// TwinCAT 3 PLC project MagnetSystem_PI4
// ProgramVersion: 3.1.4023.0
// libraries:
//   CanItfHelper, * (Beckhoff Automation LLC)
//   Tc2_Math, * (Beckhoff Automation GmbH)
//   Tc2_Standard, * (Beckhoff Automation GmbH)
//   Tc2_System, * (Beckhoff Automation GmbH)
//   Tc2_TcpIp, * (Beckhoff Automation GmbH)
//   Tc2_Utilities, * (Beckhoff Automation GmbH)
//   Tc3_Module, * (Beckhoff Automation GmbH)
//   Tc3_EventLogger,3.1.30.0,Beckhoff Automation GmbH
// project tree:
//   DUTs/ E_Command.TcDUT, E_MagState.TcDUT (not stored), E_Status.TcDUT (not stored), ST_Alarm_Base.TcDUT, ST_canRxdata.TcDUT, ST_Coil_Base.TcDUT, ST_Coil_Ext_Analog1.TcDUT, ST_Control.TcDUT, ST_EngVal.TcDUT (not stored), ST_InstFeedback.TcDUT, ST_RecipeLocal.TcDUT, ST_Setpoints.TcDUT (not stored), ST_PermissivesToMainPLC.TcDUT, ST_Recipe.TcDUT (not stored), ST_SysParameters.TcDUT (not stored), ST_Trip_Base.TcDUT, ST_UC_Status.TcDUT (not stored), ST_UC_Status_Dummy.TcDUT (not stored), ST_UCDevices.TcDUT (not stored), ST_UC_Trip_Base.TcDUT (not stored)
//   GVLs/ Alarms_DB.TcGVL, Command.TcGVL, Devices.TcGVL (not stored), HMI_DB.TcGVL (not stored), Input.TcGVL (not stored), GVL.TcGVL (not stored), InstrumentReading.TcGVL (not stored), IO.TcGVL, MCP_IO.TcGVL (not stored), Output.TcGVL, Permissives_DB.TcGVL, Recipe.TcGVL, Setpoints.TcGVL (not stored), Trips_DB.TcGVL (not stored), Tx_Config.TcGVL
//   / PlcTask.TcTTO (not stored)
//   POUs/ ADC_10V.TcPOU (not stored), ADC_5V.TcPOU (not stored), Alias.TcPOU (not stored), AnalogConversion.TcPOU, CanInterface.TcPOU (not stored), CAN_comm.TcPOU (not stored), ChargeTimeCal.TcPOU, Delay2s.TcPOU (not stored), Graphs.TcPOU, Heartbeat.TcPOU, HMI.TcPOU, MAIN.TcPOU, MODE_SELECTION_1.TcPOU, Norm_x.TcPOU (not stored), Permissives.TcPOU, ChargeRlyClose_ChargerON_Seq.TcPOU (not stored), PWMO.TcPOU, Trips.TcPOU, Tx_MasterPLC.TcPOU (not stored), VoltageOutputCal.TcPOU
// real-time tasks:
//   TASK PlcTask: cycle T#10ms, priority 20, ADS port 350

// ---- DUTs/E_Command.TcDUT
{attribute 'qualified_only'}
{attribute 'strict'}
{attribute 'to_string'}
//Command from Master PLC
TYPE E_Command :
(
	//Requested Magnetic State
	FULL_SHUTDOWN 	:= 0, 
	IDLE			:= 1, 
	CHARGE			:= 3, 
	//PAUSE_CHARGE	:= 4, //no need to use pause charge
	SHOOT			:= 6, 
	//SHUTDOWN		:= 8, //remove
	DUMP			:= 9
);
END_TYPE

// ---- DUTs/ST_Alarm_Base.TcDUT
TYPE ST_Alarm_Base :
STRUCT
(*
	AI_CH1_UnderVoltage		: BOOL;
	AI_CH1_OverVoltage		: BOOL;
	AI_CH1_belowLIM1		: BOOL;
	AI_CH1_aboveLIM1		: BOOL;
	
	AI_CH2_UnderVoltage		: BOOL;
	AI_CH2_OverVoltage		: BOOL;
	AI_CH2_belowLIM1		: BOOL;
	AI_CH2_aboveLIM1		: BOOL;
	
	AI_CH3_UnderVoltage		: BOOL;
	AI_CH3_OverVoltage		: BOOL;
	AI_CH3_belowLIM1		: BOOL;
	AI_CH3_aboveLIM1		: BOOL;
	
	ChargerVoltageReading_Faulted	: BOOL;
	CurrentReading_Faulted		 	: BOOL;
	BfieldReading_Faulted			: BOOL;
*)
	AlarmWord : WORD;
END_STRUCT
END_TYPE

// ---- DUTs/ST_canRxdata.TcDUT
TYPE ST_canRxdata :
STRUCT
	cobID			: STRING;
	deviceID		: ARRAY [1..10] OF STRING; // will make it 1..10 later
	byteData		: ARRAY [0..7] OF USINT;
	byteData_hexstr	: ARRAY [0..7] OF STRING;
END_STRUCT
END_TYPE

// ---- DUTs/ST_Coil_Base.TcDUT
//Base coil type with all the Common functionality
TYPE ST_Coil_Base :
STRUCT
	afterShot_actualCoilCurrent_WaveForm	: WORD;
	requiredTimeToCharge					: TIME;
	measuredMagneticField					: DINT;
		
	ChargeVoltageFeedback					: REAL;
	ChargeVoltageFeedback_raw				: INT;
	ChargerVoltageFeedback_norm				: REAL;
	TotalVoltage							: REAL;
	
	CurrentFeedback							: REAL;
	CurrentFeedback_raw						: INT;
	CurrentFeedback_norm					: REAL;

	Measured_Bfield							: REAL;
	Measured_Bfield_raw						: INT;
	B_fieldFeedback_norm					: REAL;
	
	chargerSetpoint							: INT;  //0-100% analog PWM 24V output -> (0 - 10V)
	chargerSetpoint_norm					: REAL;
	chargerSetpoint_raw						: REAL;
	currentSetpoint							: INT;  //0-100% analog PWM 24V output -> (0.5 - 4.5V)
	currentSetpoint_norm					: REAL;
	currentSetpoint_raw						: REAL;
	//currentSetpointFromMaster: REAL;

	PSU0_active								: BOOL := FALSE;
	PSU1_DCOK								: BOOL;
	Local_StopPB_Pressed					: BOOL;  //NC
	DumpRelay1_closed						: BOOL;
	DumpRelay2_closed						: BOOL;
	ChargeRelay_closed						: BOOL := FALSE;
	ChargerIsEnabled						: BOOL := FALSE; //feedback from charger
	FlybackD1_Alive							: BOOL := FALSE;
	FlybackD2_Alive							: BOOL := FALSE;
	
	DumpResistorTemperatureHigh				: BOOL; 
	GroundLoopCurrentDetected				: BOOL;
	CoilTemperatureHigh						: BOOL := FALSE;
	AC_Interlock_RlyClose					: BOOL;
	LossPneumaticPressure					: BOOL;
	
	OpenDumpRelays							: BOOL := FALSE;
	closeChargeRelay						: BOOL := FALSE;
	enableOutputToCharger					: BOOL := FALSE;  //output going to charger
	CloseACInterlockRly						: BOOL := FALSE;
	SystemFaulted							: BOOL := FALSE;
	SystemCharging							: BOOL := FALSE;
	SystemReady								: BOOL := FALSE;
	CloseHVisolationRelay					: BOOL; //relay 6 (24vdc) to control relay 7 & 8 (two 120vac ross relays)
	HVisolationRelayClosed					: BOOL;
	OutputRelayOpen							: BOOL;
	
	CoilEnabled								: BOOL := TRUE;
	AllCapsCharged							: BOOL;
	NumOfCap								: INT := 4;
	
	//CoilSafetyOK							: BOOL;
	CapWarning								: BOOL;  //comes from UltraCaps CANBUS message
	CapAlarm								: BOOL;
	CapVoltage								: ARRAY[1..15] OF INT;   //Comes from UlgraCaps CANBUS message
	CapCellTemp								: ARRAY[1..15] OF INT;
	
	ChargerVoltageFault_TON : TON;
	ChargerVoltageFault_ET : TIME;
	CurrentSensorFault_TON : TON;
	CurrentSensorFault_ET : TIME;
	BfieldSensorFault_TON : TON;
	BfieldSensorFault_ET : TIME;
	
	//CAN_id: INT;
	//CAN_AdsAddr: AMSADDR;
	//CAN_netID: AMSNETID;
	//CAN_port: WORD;
	//CAN_error: USINT;
	//CAN_State: UINT;
	//CAN_RxErrorCounter: USINT;	
	//CAN_TxErrorCounter: USINT;	
	//CAN_DiagFlag: BOOL;
	
	//UltraCap_CAN_ID : STRING;
	UltraCap			: ARRAY[1..10] OF  ST_UC_Status;  //assuming 10 uc in one coil
	UltraCap_Dummy		: ST_UC_Status_Dummy; //buffer temp for uc 7f
	UC_Dummy_ID_hexstr	: STRING;
	
	CanTx_config_ID 	: UDINT;
	CanTx_config_length : UINT;
	CanTx_config_request: ARRAY[0..7] OF BYTE;
		
END_STRUCT
END_TYPE

// ---- DUTs/ST_Coil_Ext_Analog1.TcDUT
TYPE ST_Coil_Ext_Analog1 EXTENDS ST_Coil_Base :
STRUCT
	iAnalogOfWinning : INT;
END_STRUCT
END_TYPE

// ---- DUTs/ST_Control.TcDUT
TYPE ST_Control :
STRUCT
	ClearAllFault : BOOL;
	Abort		  : BOOL;
END_STRUCT
END_TYPE

// ---- DUTs/ST_InstFeedback.TcDUT
TYPE ST_InstFeedback :
STRUCT
	ChargerVolt : REAL;
	CapVolt		: ARRAY [1..15] OF REAL;
	Cur  		: REAL;
	TotalVoltage: REAL;
END_STRUCT
END_TYPE

// ---- DUTs/ST_RecipeLocal.TcDUT
TYPE ST_RecipeLocal :
STRUCT
	chargerSetpoint 	: INT;  
	currentSetpoint 	: INT;   
	CurrentDuration		: TIME;   
END_STRUCT
END_TYPE

// ---- DUTs/ST_PermissivesToMainPLC.TcDUT
TYPE ST_PermissivesToMainPLC :
STRUCT
	ChargePermOK			: BOOL;
	ShootPermOK				: BOOL;
	
	AlldcPSUok				: BOOL;
	AllacInterlock_Closed	: BOOL;
	All_Coil_TemperatureOK	: BOOL;
	AllDumpResistorTempOK	: BOOL;
	NoGroundLoopCurrentDetected: BOOL;
	//AllFlybackDiodes_Alive	: BOOL;
	AllChargerEnabled		: BOOL;
	AnyCoilDisabled 		: BOOL;		
	SafetyOK				: BOOL;
	AllDumpRelayOpen		: BOOL;
	AllChargerRelay_Closed	: BOOL;
	AdminFaultBypassOn		: BOOL;
	// voltage feedback from CANbus to main plc
	
END_STRUCT
END_TYPE

// ---- DUTs/ST_Trip_Base.TcDUT
TYPE ST_Trip_Base :
STRUCT
	ChargerVoltageReadingFaulted 		: BOOL;
	CurrentReadingFaulted 		 		: BOOL;
	BfieldReadingFaulted 		 		: BOOL;
	
	ACInterlockRelayFailedtoClose		: BOOL;
	ACInterlockRelayFailedtoOpen 		: BOOL;
	ACintLockRlyCloseFaultDelay_TON		: TON;
	ACintLockRlyOpenFaultDelay_TON		: TON;
	
	DumpRelay1_FailtoClose		 		: BOOL;
	DumpRelay1_FailtoOpen		 		: BOOL;
	DumpRlyCloseFaultDelay_TON 		 	: TON;
	DumpRlyOpenFaultDelay_TON 		 	: TON;
	
	DumpRelay2_FailtoClose		 : BOOL;
	DumpRelay2_FailtoOpen		 : BOOL;
	
	ChargeRelay_FailtoClose		 : BOOL;
	ChargeRelay_FailtoOpen		 : BOOL;
	ChrgRlyCloseFaultDelay_TON	 : TON;
	ChrgRlyOpenFaultDelay_TON	 : TON;
	
	
	HVisoRelayFailedToOpen		: BOOL;
	HVRelayOpenFaultDelay_TON	: TON;
	HVisoRelayFailedToClose		: BOOL;
	HVRelayCloseFaultDelay_TON	: TON;
	
	UltraCap					: ARRAY[1..10] OF ST_UC_Trip_Base;
	AnyCapOverV_warning			: BOOL;  //cell voltage > 2.85V - warning, > 2.9V - alarm
	AnyCapOverV_alarm			: BOOL;  //cell voltage > 2.85V - warning, > 2.9V - alarm
	AnyCapOverTemp_warning		: BOOL; //cell >50C - warning, >60C - alarm
	AnyCapOverTemp_alarm		: BOOL; //cell >50C - warning, >60C - alarm
END_STRUCT
END_TYPE

// ---- GVLs/Alarms_DB.TcGVL
{attribute 'qualified_only'}
VAR_GLOBAL
	Coil1 : ST_Alarm_Base;
	Coil2 : ST_Alarm_Base;
	Coil3 : ST_Alarm_Base;
	Coil4 : ST_Alarm_Base;
	Coil5 : ST_Alarm_Base;
	Coil6 : ST_Alarm_Base;
	Coil7 : ST_Alarm_Base;
	Coil8 : ST_Alarm_Base;
	Coil9 : ST_Alarm_Base;
	Coil10 : ST_Alarm_Base;
	
	AlarmWord_11 : ST_Alarm_Base;
	AlarmWord_22 : ST_Alarm_Base;
	AlarmWord_23 : ST_Alarm_Base;
	AlarmWord_24 : ST_Alarm_Base;
	AlarmWord_25 : ST_Alarm_Base;
	AlarmWord_26 : ST_Alarm_Base;
	AlarmWord_27 : ST_Alarm_Base;
	AlarmWord_88 : ST_Alarm_Base;
END_VAR

// ---- GVLs/Command.TcGVL
{attribute 'qualified_only'}
VAR_GLOBAL

	eCommand : E_Command;
END_VAR

// ---- GVLs/IO.TcGVL
{attribute 'qualified_only'}
VAR_GLOBAL
	//PB01_Rx AT%I* : ARRAY [0..145] OF BYTE;
	//PB01_Tx AT%Q* : ARRAY [0..145] OF BYTE;
END_VAR

// ---- GVLs/Output.TcGVL
{attribute 'qualified_only'}
VAR_GLOBAL
//LCP 1	
	//EL2502 - PWM Output
	R2_02_00 AT %Q*: INT;
	R2_02_01 AT %Q*: INT;
	
	// EL 2008 - DQ
	R2_05_00 AT %Q*: BOOL;
	R2_05_01 AT %Q*: BOOL;
	R2_05_02 AT %Q*: BOOL;
	R2_05_03 AT %Q*: BOOL;
	R2_05_04 AT %Q*: BOOL;
	R2_05_05 AT %Q*: BOOL;
	R2_05_06 AT %Q*: BOOL;
	R2_05_07 AT %Q*: BOOL; //spare
	
	R2_06_CANrequest AT %Q*: EXTCANQUEUE;
//LCP 2	***********************************************
	//EL2502 - PWM Output
	R3_02_00 AT %Q*: INT;
	R3_02_01 AT %Q*: INT;
	
	// EL 2008 - DQ
	R3_05_00 AT %Q*: BOOL;
	R3_05_01 AT %Q*: BOOL;
	R3_05_02 AT %Q*: BOOL;
	R3_05_03 AT %Q*: BOOL;
	R3_05_04 AT %Q*: BOOL;
	R3_05_05 AT %Q*: BOOL;
	R3_05_06 AT %Q*: BOOL;
	R3_05_07 AT %Q*: BOOL; //spare
	
	R3_06_CANrequest AT %Q*: EXTCANQUEUE;	
END_VAR

// ---- GVLs/Permissives_DB.TcGVL
{attribute 'qualified_only'}
VAR_GLOBAL
	ChargePermOK			: BOOL;
	ShootPermOK				: BOOL;
	//AllChargers_Active		: BOOL;
	AlldcPSUok				: BOOL;
	AllacInterlock_Closed	: BOOL;
	All_Coil_TemperatureOK	: BOOL;
	AllDumpResistorTempOK	: BOOL;
	NoGroundLoopCurrentDetected: BOOL;
	//AllFlybackDiodes_Alive	: BOOL;
	AllChargerEnabled		: BOOL;
	AnyCoilDisabled 		: BOOL;		
	SafetyOK				: BOOL;
	AllDumpRelayOpen		: BOOL;
	//AllDumpRelayClose		: BOOL;
	AllChargerRelay_Closed	: BOOL;
	AllCoilCapsCharged		: BOOL;
	NoPneumaticPressureLoss : BOOL;
END_VAR

// ---- GVLs/Recipe.TcGVL
{attribute 'qualified_only'}
VAR_GLOBAL
	Coil : ARRAY[1..10] OF ST_Recipe;
	General : ST_Recipe;
END_VAR

// ---- GVLs/Tx_Config.TcGVL
{attribute 'qualified_only'}
VAR_GLOBAL
	CoilSP : ARRAY[1..10] OF ST_Setpoints;
	
	ReadyToChargeRunOutTime	: REAL;
	ChargingRunOutTime		: REAL;
	ChargePausedRunOutTime	: REAL;
	ReadyToShootRunOutTime	: REAL;				
	ShootingRunOutTime		: REAL;
	PostShotRunOutTime		: REAL;
	DumpingRunOutTime		: REAL;
	CoilInst				: ARRAY[1..10] OF ST_InstFeedback;
	
END_VAR

// ---- POUs/AnalogConversion.TcPOU
PROGRAM AnalogConversion
VAR	
	i : INT  := 1;
	
END_VAR

//*******************Output Sepoints come from the Screen room recipe, the sysparameters would need to mapped here******//
//ie Setpoints.coil[1].engval.max_chargervoltage := Recipe.
Devices.Coil[1].NumOfCap := Setpoints.Coil[1].SysParameters.NumOfCaps;


//Converting raw data into Voltage Reading (0-10V), (0.5-4.5V)

//LCP1
// Voltage feedback - 10V = Max voltage (102V)
Devices.Coil[1].ChargerVoltageFeedback_norm := Norm_x (raw_input := INT_TO_REAL(Devices.Coil[1].ChargeVoltageFeedback_raw),
										x_max := 32767,
										x_min := 0);
										
InstrumentReading.R2_01_CH00 := Devices.Coil[1].ChargerVoltageFeedback_norm * 10;

//Charger Voltage = (max voltage - min voltage) * measured_voltage / range(voltage)
Devices.Coil[1].ChargeVoltageFeedback := (Setpoints.Coil[1].EngVal.Max_chargerVoltage - Setpoints.Coil[1].EngVal.Min_chargerVoltage) * ADC_10V (normal_input := Devices.Coil[1].ChargerVoltageFeedback_norm,
																					x_max := 10,
																					x_min := 0);

//Current feedback - 4.5V = 600Amp????
Devices.Coil[1].CurrentFeedback_norm := Norm_x (raw_input := INT_TO_REAL(Devices.Coil[1].CurrentFeedback_raw),
								x_max := 32767*4.5/10,
								x_min := 32767*0.5/10);
						
InstrumentReading.R2_01_CH01 := Devices.Coil[1].CurrentFeedback_norm * (4.5-0.5);

//Current feedback for each ultracap
Devices.Coil[1].CurrentFeedback := (Setpoints.Coil[1].EngVal.Max_current_perCap - Setpoints.Coil[1].EngVal.Min_current_perCap) * ADC_5V (normal_input := Devices.Coil[1].CurrentFeedback_norm,
																								x_max := 4.5,
																								x_min := 0.5);

//CurrentFeedback_norm := Norm_x (raw_input := INT_TO_REAL(Input.R2_01_01), x_max := 32767*4.5/10, x_min := 32767*0.5/10);
//coil1.CurrentFeedback := CurrentFeedback_norm * 4;

//B-field - (0-10V) 10V = ?? Tesla
Devices.Coil[1].B_fieldfeedback_norm := Norm_x (raw_input := INT_TO_REAL(Devices.Coil[1].Measured_Bfield_raw),
								x_max := 32767,
								x_min := 0);
								
InstrumentReading.R2_01_CH02 := Devices.Coil[1].B_fieldfeedback_norm * 10;

//Charger Voltage = (max voltage - min voltage) * measured_voltage / range(voltage)
Devices.Coil[1].Measured_Bfield := (Setpoints.Coil[1].EngVal.Max_Tesla - Setpoints.Coil[1].EngVal.Min_Tesla) * ADC_10V(normal_input := Devices.Coil[1].B_fieldfeedback_norm,
																x_max := 10,
																x_min := 0);

																
//PWM Output

//set limits of charger voltage input 
FOR i := 1 TO 10 BY 1 DO
	IF Devices.Coil[i].chargerSetpoint >= REAL_TO_INT (Setpoints.Coil[1].EngVal.Max_chargerVoltage) THEN
		Devices.Coil[i].chargerSetpoint := REAL_TO_INT (Setpoints.Coil[1].EngVal.Max_chargerVoltage);
	END_IF;
	//This should never happend
	IF Devices.Coil[i].chargerSetpoint_raw >= (10/24 * 32767) THEN
		Devices.Coil[i].chargerSetpoint_raw := (10/24 * 32767);
	END_IF;
END_FOR;

Devices.Coil[1].chargerSetpoint_norm := Norm_x (raw_input := INT_TO_REAL (Devices.Coil[1].chargerSetpoint), 
												x_max := Setpoints.Coil[1].EngVal.Max_chargerVoltage,
												x_min := Setpoints.Coil[1].EngVal.Min_chargerVoltage);

Devices.Coil[1].chargerSetpoint_raw := PWMO (norm_input := Devices.Coil[1].chargerSetpoint_norm, 
												x_max := 24,
												x_min := 0); 	


//Current set point output
//set limits of charger voltage input 
FOR i := 1 TO 10 BY 1 DO
	IF Devices.Coil[i].currentSetpoint >= REAL_TO_INT (Setpoints.Coil[1].EngVal.Max_current_perCap) THEN
		Devices.Coil[i].currentSetpoint := REAL_TO_INT (Setpoints.Coil[1].EngVal.Max_current_perCap);
	END_IF;
	//This should never happend - Current setpoint board takes 0.5V - 4.5V
	IF Devices.Coil[i].currentSetpoint_raw >= (4.5/24 * 32767) THEN
		Devices.Coil[i].currentSetpoint_raw := (4.5/24 * 32767);
	END_IF;
END_FOR;

Devices.Coil[1].currentSetpoint_norm := Norm_x (raw_input := INT_TO_REAL (Devices.Coil[1].currentSetpoint), 
												x_max := Setpoints.Coil[1].EngVal.Max_current_perCap,
												x_min := Setpoints.Coil[1].EngVal.Min_current_perCap);
//current output for each cap
Devices.Coil[1].currentSetpoint_raw := PWMO (norm_input := Devices.Coil[1].currentSetpoint_norm, 
												x_max := 24,
												x_min := 0); 	


//uncomment this when PWM output module is ready.											
(*
//LCP1
Output.R2_02_00 := Devices.Coil[1].chargerSetpoint_raw; 
Output.R2_02_01 := Devices.Coil[1].currentSetpoint_raw;

//LCP2
Output.R3_02_00 := Devices.Coil[2].chargerSetpoint_raw; 
Output.R3_02_01 := Devices.Coil[2].currentSetpoint_raw;
*)

//reset counter
IF i > 10 THEN
	i:=1;
END_IF;

END_PROGRAM

// ---- POUs/PWMO.TcPOU
FUNCTION PWMO : INT
VAR_INPUT
	Norm_input : REAL;
	x_max : REAL := 24;
	x_min : REAL := 0;
END_VAR
VAR
	voltage_reading : REAL;
END_VAR

voltage_reading := 10 * Norm_input;
PWMO := REAL_TO_INT (32767 * (voltage_reading - x_min) / (x_max - x_min));

END_FUNCTION

// ---- POUs/ChargeTimeCal.TcPOU
FUNCTION_BLOCK ChargeTimeCal
VAR_INPUT
	I_setpoint 	: REAL := 400;
	t_duration	: REAL := 4;
	NumOfCaps	: REAL := 15;
	C_percap	: REAL := 88;
	VMAXperCap	: REAL := 100;
	R_coil		: REAL := 1.1;
	L_coil		: REAL := 0.5;
	VMAXcharger	: REAL := 1500;
	Pcharger	: REAL := 15000;
	NumOfCharger: REAL := 4;
END_VAR
VAR_OUTPUT
	Tuntilfullcharge	: REAL;
END_VAR
VAR
	V_chargerCC2CP : REAL;
	C_total		   : REAL;
	V_capsmax	   : REAL;
	E_resistivepulse : REAL;
	E_inductivepulse : REAL;
	E_pulse			 : REAL;
	VchrSPrequested  : REAL;
	VchrSPactual     : REAL;
	I_peakchargecurrent : REAL;
	Icc					: REAL;
	Icp					: REAL;
	Vpresent			: REAL;
	Vfinal				: REAL;
	VpresentCC			: REAL;
	VfinalCC			: REAL;
	Tcc					: REAL;
	VpresentCP			: REAL;
	Tcp					: REAL;
END_VAR

V_chargerCC2CP := VMAXcharger / 2;

C_total := C_percap/NumOfCaps;
V_capsmax := VMAXpercap * NumOfCaps;
E_resistivepulse := LREAL_TO_REAL(EXPT(I_setpoint, 2))*R_coil*t_duration;
E_inductivepulse := L_coil * LREAL_TO_REAL(EXPT(I_setpoint, 2))/2;
E_pulse := E_resistivepulse + E_inductivepulse;
VchrSPrequested := SQRT(2*E_pulse/C_total);

IF VchrSPrequested > V_capsmax THEN
	VchrSPactual := V_capsmax;
	ELSE
		VchrSPactual := VchrSPrequested;	
END_IF

//I_peakchargecurrent := Pcharger * NumOfCharger / (2*VMAXcharger);
I_peakchargecurrent := Pcharger * NumOfCharger * 2 / VMAXcharger;
Icc := I_peakchargecurrent;
Icp := I_peakchargecurrent * (0.5 + ((VMAXcharger - Vpresent)/VMAXcharger));
Vfinal := 1400; //hard coded???
VpresentCC := 200; // hard coded???

IF Vfinal > V_chargerCC2CP THEN
	VfinalCC := V_chargerCC2CP;
	ELSIF Vfinal < V_chargerCC2CP THEN
		VfinalCC := Vfinal;
END_IF

Tcc := (V_chargerCC2CP - VpresentCC)*C_total/I_peakchargecurrent;

VpresentCP := V_chargerCC2CP;
Tcp := -((VMAXcharger*C_total)/I_peakchargecurrent)*LN((1.5*VMAXcharger-Vfinal)/(1.5*VMAXcharger-VpresentCP));

Tuntilfullcharge := Tcc + Tcp;

END_FUNCTION_BLOCK

// ---- POUs/Graphs.TcPOU
PROGRAM Graphs
VAR
	i : INT :=0;
	coil1_current: ARRAY[1..1, 1..100] OF REAL;
	//coil1_current : ARRAY	

END_VAR

// still need more work

FOR i := 1 TO 100 DO 
	coil1_current[1, i] := Devices.coil1.CurrentFeedback;
	
END_FOR

FOR i := 100 TO 2 BY -1 DO
	coil1_current[1, i-1] := Devices.coil1.CurrentFeedback;
END_FOR

IF coil1_current[1, 1] = 100 THEN
	i := -1;
ELSIF coil1_current[1, 1] = 1 THEN
	i := 1;
END_IF

END_PROGRAM

// ---- POUs/Heartbeat.TcPOU
PROGRAM Heartbeat
VAR
	start_TON				: TON;
	start_TON_et 			: TIME;
	reset_TON 				: TON;
	reset_TON_et 			: TIME;
	screen_refresh_pulse 	: BOOL;
	
	pulse_1Hz_Start_TON		: TON;
	pulse_1Hz_Start_PT		: TIME := T#4MS;
	pulse_1Hz_Reset_TON		: TON;
	pulse_1Hz_Reset_PT		: TIME := T#6MS;
	pulse_1Hz				: BOOL;
END_VAR

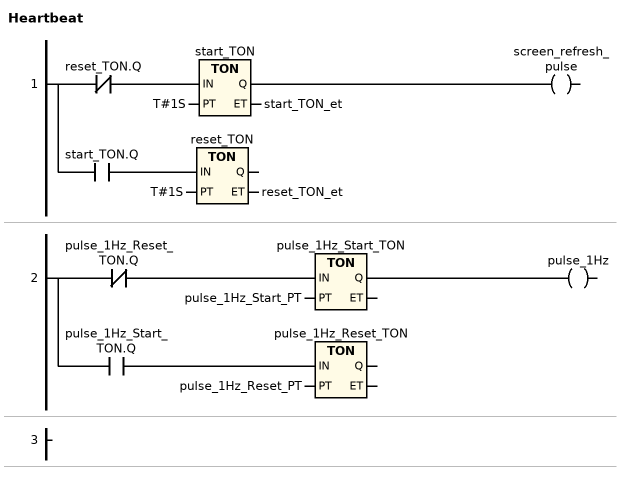
// NETWORK 1
start_TON(IN := NOT reset_TON.Q, PT := T#1S, ET => start_TON_et); // TON
screen_refresh_pulse := start_TON.Q;
reset_TON(IN := start_TON.Q, PT := T#1S, ET => reset_TON_et); // TON

// NETWORK 2
pulse_1Hz_Start_TON(IN := NOT pulse_1Hz_Reset_TON.Q, PT := pulse_1Hz_Start_PT); // TON
pulse_1Hz := pulse_1Hz_Start_TON.Q;
pulse_1Hz_Reset_TON(IN := pulse_1Hz_Start_TON.Q, PT := pulse_1Hz_Reset_PT); // TON

// NETWORK 3

END_PROGRAM

// ---- POUs/HMI.TcPOU
PROGRAM HMI
VAR
END_VAR



HMI_DB.ReadyToChargeRunOutTime	:= TIME_TO_DINT (MODE_SELECTION_1.ReadyToChargeRunOutTMR_PT - MODE_SELECTION_1.ReadyToChargeRunOutTMR_TON.ET)/1000;
HMI_DB.ChargingRunOutTime		:= TIME_TO_DINT (MODE_SELECTION_1.ChargingRunOutTMR_PT - MODE_SELECTION_1.ChargingRunOutTMR_TON.ET)/1000;	
HMI_DB.ChargePausedRunOutTime	:= TIME_TO_DINT (MODE_SELECTION_1.ChargePausedRunOutTMR_PT - MODE_SELECTION_1.ChargePausedRunOutTMR_ET)/1000;	
HMI_DB.ReadyToShootRunOutTime	:= TIME_TO_DINT (MODE_SELECTION_1.ReadyToShootRunOutTMR_PT - MODE_SELECTION_1.ReadyToShootRunOutTMR_ET)/1000;					
HMI_DB.ShootingRunOutTime		:= TIME_TO_DINT (MODE_SELECTION_1.ShootingRunOutTMR_PT - MODE_SELECTION_1.ShootingRunOutTMR_ET)/1000;			
HMI_DB.PostShotRunOutTime		:= TIME_TO_DINT (MODE_SELECTION_1.PostShotRunOutTMR_PT - MODE_SELECTION_1.PostShotRunOutTMR_ET)/1000;			
HMI_DB.DumpingRunOutTime		:= TIME_TO_DINT (MODE_SELECTION_1.DumpingRunOutTMR_PT - MODE_SELECTION_1.DumpingRunOutTMR_ET)/1000;

END_PROGRAM

// ---- POUs/MODE_SELECTION_1.TcPOU
PROGRAM MODE_SELECTION_1
VAR
	//MagnetState : (FULL_SHUTDOWN, IDLE, READY_TO_CHARGE, CHARGING, CHARGING_PAUSED, READY_TO_SHOOT, SHOOTING, POST_SHOT, SHUTDOWN, DUMPING); 
	eMagState : E_MagState := 0;
	//bChargingDone: BOOL;
	eCommand : E_Command; // Requested State (FULL_SHUT_DOWN = 0, IDLE = 1, CHARGE = 2, CHARGE_PAUSED, SHOOT = 3, POST_SHOT = 4, SHUTDOWN = 5, DUMPING = 6)
	eStatus : E_Status; // Actual Status (FULL_SHUTDOWN = 0, IDLE = 1, READY_TO_CHARGE = 2, CHARGE = 3, CHARGE_PAUSED = 4, READY_TO_SHOOT = 5, SHOOTING = 6, POST_SHOT = 7, SHUTDOWN = 8, DUMPING = 9, TRIPPED = 10, MANUAL_MODE = 11)
	i: INT;
	
	ChargerOFF_ChrgRlyOPEN_Delay_FShutDown_TON	: TON;
	timerBTW_ChrgRly_ChrgEnable_ChrgPause_TON	: TON;
	timerBTW_ChrgRly_ChrgEnable_ReadyToShoot_TON: TON;
	
	timerBTW_ChrgRly_ChrgEnable_Chrging_TON		: TON;
	timerBTW_ChrgRly_ChrgEnable_PT 	: TIME := T#500MS;
	timerBTW_ChrgRly_ChrgEnable_ET  : TIME;
	
	timerBTW_DUMP_IDLE 				: TON;
	timerBTW_DUMP_IDLE_PT 			: TIME := T#15S;
	timerBTW_DUMP_IDLE_ET 			: TIME;
	
	timerForChargertoTurnOn_TON		: TON;
	timerForChargertoTurnOn_PT		: TIME := T#10S;
	timerForChargertoTurnOn_ET		: TIME;
	ChargersReady					: BOOL;
	
	timerBTW_Shoot_PostShot_TON		: TON;
	timerBTW_Shoot_PostShot_PT      : TIME := T#2S;
	timerBTW_Shoot_PostShot_ET		: TIME;
	
	timerBTW_ChrgEnable_ChrgRly_ShutDown_TON	: TON;
	timerBTW_ChrgEnable_ChrgRly_PT				: TIME := T#1S;
	timerBTW_ChrgEnable_ChrgRly_ET				: TIME;
	
	timerBTW_ChrgEnable_ChrgRly_Dumping_TON		: TON;
	timerBTW_ChrgEnable_ChrgRly_Dumping_ET		: TIME;
	
	timerBTW_ChrgEnable_ChrgRly_Tripped_TON		: TON;
	timerBTW_ChrgEnable_ChrgRly_Tripped_ET		: TIME;
	
	ReadyToChargeRunOutTMR_TON					: TON;
	ReadyToChargeRunOutTMR_PT					: TIME := T#1200S;
	ReadyToChargeRunOutTMR_ET					: TIME;
	
	ChargePausedRunOutTMR_TON					: TON;
	ChargePausedRunOutTMR_PT					: TIME := T#30S;
	ChargePausedRunOutTMR_ET					: TIME;
	
	ReadyToShootRunOutTMR_TON					: TON;
	ReadyToShootRunOutTMR_PT					: TIME := T#60S;
	ReadyToShootRunOutTMR_ET					: TIME;
	
	ShootingRunOutTMR_TON						: TON;
	ShootingRunOutTMR_PT						: TIME := T#3S;
	ShootingRunOutTMR_ET						: TIME;
	
	PostShotRunOutTMR_TON						: TON;
	PostShotRunOutTMR_PT						: TIME := T#2S;
	PostShotRunOutTMR_ET						: TIME;
	
	DumpingRunOutTMR_TON						: TON;
	DumpingRunOutTMR_PT							: TIME := T#300S;
	DumpingRunOutTMR_ET							: TIME;
	
	ChargingRunOutTMR_TON						: TON;
	ChargingRunOutTMR_PT						: TIME := T#600S;
	ChargingRunOutTMR_ET						: TIME;
	
	stControl									: ST_Control;
END_VAR


//LCP Indicator for charged/charging
FOR i := 1 TO 10 BY 1 DO
	IF ( Devices.Coil[i].ChargeRelay_closed = TRUE AND 
		Devices.Coil[i].CoilEnabled = TRUE AND 
		Devices.Coil[i].enableOutputToCharger = TRUE ) OR Devices.Coil[i].ChargeVoltageFeedback >= 10
	THEN
		Devices.Coil[i].SystemCharging := TRUE;
		ELSE
			Devices.Coil[i].SystemCharging := FALSE;
	END_IF;
END_FOR;

//IF any one of the systems is charging or charge, then all system discharge is false, otherwise true
IF Devices.Coil[i].SystemCharging = TRUE THEN
	GVL.AllSystemsDischarged := FALSE;
ELSE
	GVL.AllSystemsDischarged := TRUE;
END_IF;

// IF system is tripped at anytime, it goes to tripped state
IF Trips_DB.SystemTripped = TRUE OR Permissives_DB.SafetyOK = FALSE THEN
	eMagState := E_MagState.TRIPPED;
END_IF;

IF MCP_IO.RemoteModeSelected = FALSE OR HMI_DB.RemoteModeSelected = FALSE THEN  //change auto to remote / manu to local
	eStatus := E_Status.MANUAL_MODE;
END_IF

//At any point, if screen room ask to dump, it goes to dump state
IF (MCP_IO.RemoteModeSelected = TRUE AND eCommand = E_Command.DUMP) OR stControl.Abort = TRUE THEN
	eMagState := E_Magstate.DUMPING;
END_IF;

FOR i := 1 TO 10 BY 1 DO
	Devices.Coil[i].NumOfCap := Tx_Config.CoilSP[i].SysParameters.NumOfCaps;
END_FOR


//Process Starts
CASE eMagState OF 
	//Full Shutdown
	E_MagState.FULL_SHUTDOWN:
						//Disable all Chargers
						FOR i := 1 TO 10 BY 1 DO
							
							//open (de-energize) all interlock relays
							Devices.Coil[i].CloseACInterlockRly := FALSE;
							Devices.Coil[i].enableOutputToCharger := FALSE;
			
							//Close (de-energize) All Dump relays
							Devices.Coil[i].OpenDumpRelays := FALSE;
							
							Devices.Coil[i].CloseHVisolationRelay := FALSE;   //Open all HV isolation relays
						END_FOR;
						
						ChargerOFF_ChrgRlyOPEN_Delay_FShutDown_TON (IN:=TRUE, PT:= timerBTW_ChrgRly_ChrgEnable_PT);
						//delay 500ms before opening charge relay
						IF ChargerOFF_ChrgRlyOPEN_Delay_FShutDown_TON.Q = TRUE THEN
							FOR i := 1 TO 10 BY 1 DO		
							//open (de-energize) all interlock relays
							Devices.Coil[i].closeChargeRelay := FALSE;	
							END_FOR;
							ChargerOFF_ChrgRlyOPEN_Delay_FShutDown_TON (IN:=FALSE, PT:= timerBTW_ChrgRly_ChrgEnable_PT);
						END_IF;
						
						//send shutdown status to screen room
						eStatus := E_Status.FULL_SHUTDOWN;
						//if auto mode selected or hmi automode is selected and screen room asks for idle mode go to idle mode
						IF (MCP_IO.RemoteModeSelected = TRUE OR HMI_DB.RemoteModeSelected = TRUE) AND eCommand = E_Command.IDLE THEN //Auto mode
							GVL.fullshutdown_to_idle := TRUE;
							//if in manu mode and safety is okay and HMI idle MODE PB is pressed, go to idle mode
						ELSIF HMI_DB.RemoteModeSelected = FALSE AND Permissives_DB.SafetyOK = TRUE AND HMI_DB.Idle_mode = TRUE THEN //Manu mode
							GVL.fullshutdown_to_idle := TRUE;
						ELSE
							GVL.fullshutdown_to_idle := FALSE; // otherwise do nothing.
						END_IF;
	
						IF GVL.fullshutdown_to_idle = TRUE THEN
							eMagState := E_MagState.IDLE;
						END_IF;
						//reset all run out tmr
						ReadyToChargeRunOutTMR_TON (IN := FALSE, PT := ReadyToChargeRunOutTMR_PT, ET=>ReadyToChargeRunOutTMR_ET);
						ChargingRunOutTMR_TON (IN := FALSE, PT := ChargingRunOutTMR_PT, ET => ChargingRunOutTMR_ET);
						ChargePausedRunOutTMR_TON (IN := FALSE, PT := ChargePausedRunOutTMR_PT, ET=> ChargePausedRunOutTMR_ET);
						ReadyToShootRunOutTMR_TON (IN := FALSE, PT := ReadyToShootRunOutTMR_PT, ET => ReadyToShootRunOutTMR_ET);
						ShootingRunOutTMR_TON (IN := FALSE, PT := ShootingRunOutTMR_PT, ET => ShootingRunOutTMR_ET);
						PostShotRunOutTMR_TON (IN := FALSE, PT := PostShotRunOutTMR_PT, ET => PostShotRunOutTMR_ET);
						DumpingRunOutTMR_TON (IN := FALSE, PT := DumpingRunOutTMR_PT, ET => DumpingRunOutTMR_ET);
		
	//IDLE STATE
	E_MagState.IDLE:
						eStatus := E_Status.IDLE; //Send status state to screen room
						GVL.dump_to_idle := FALSE;
						//reset all run out tmr
						ReadyToChargeRunOutTMR_TON (IN := FALSE, PT := ReadyToChargeRunOutTMR_PT, ET=>ReadyToChargeRunOutTMR_ET);
						ChargingRunOutTMR_TON (IN := FALSE, PT := ChargingRunOutTMR_PT, ET => ChargingRunOutTMR_ET);
						ChargePausedRunOutTMR_TON (IN := FALSE, PT := ChargePausedRunOutTMR_PT, ET=> ChargePausedRunOutTMR_ET);
						ReadyToShootRunOutTMR_TON (IN := FALSE, PT := ReadyToShootRunOutTMR_PT, ET => ReadyToShootRunOutTMR_ET);
						ShootingRunOutTMR_TON (IN := FALSE, PT := ShootingRunOutTMR_PT, ET => ShootingRunOutTMR_ET);
						PostShotRunOutTMR_TON (IN := FALSE, PT := PostShotRunOutTMR_PT, ET => PostShotRunOutTMR_ET);
						DumpingRunOutTMR_TON (IN := FALSE, PT := DumpingRunOutTMR_PT, ET => DumpingRunOutTMR_ET);
						
						// Local MODE
						IF (MCP_IO.RemoteModeSelected = FALSE OR HMI_DB.RemoteModeSelected = FALSE)AND 
							HMI_DB.chargePB = TRUE AND 
							Permissives_DB.SafetyOK = TRUE AND 
							GVL.AllSystemsDischarged = TRUE 
							THEN   
								//open dump relays
								FOR i := 1 TO 10 BY 1 DO
									Devices.Coil[i].OpenDumpRelays := TRUE; //NC contact
								END_FOR;
			
								GVL.idle_to_readyToCharge := TRUE;
							ELSE
								GVL.idle_to_readyToCharge := FALSE;
						END_IF;
						//Remote MODE
						// ready to go to charge state when dump relays are all open and charge permissive is satisfied 
						IF (MCP_IO.RemoteModeSelected = TRUE OR HMI_DB.RemoteModeSelected = TRUE) AND 
							Permissives_DB.SafetyOK = TRUE AND GVL.AllSystemsDischarged = TRUE
							THEN 
								//open dump relays
								FOR i := 1 TO 10 BY 1 DO
									Devices.Coil[i].OpenDumpRelays := TRUE; //NC contact
								END_FOR;	
								GVL.idle_to_readyToCharge := TRUE;
						ELSE
							GVL.idle_to_readyToCharge := FALSE;
							//Keep dump relays close if no command to go to charging state
							FOR i := 1 TO 10 BY 1 DO
								Devices.Coil[i].OpenDumpRelays := FALSE; //NC contact
							END_FOR;
						END_IF;
		
						IF GVL.idle_to_readyToCharge = TRUE AND Permissives_DB.ChargePermOK = TRUE AND GVL.AllSystemsDischarged = TRUE THEN
							eMagState := E_MagState.READY_TO_CHARGE;
						ELSIF (MCP_IO.RemoteModeSelected = TRUE AND eCommand = E_Command.FULL_SHUTDOWN) 
							THEN 
								eMagState := E_MagState.FULL_SHUTDOWN;
						END_IF;
						
	//Charging State	
	E_MagState.READY_TO_CHARGE:
						//reset bit
						GVL.idle_to_readyToCharge := FALSE;
						//send status to screenroom
						eStatus := E_Status.READY_TO_CHARGE;
						
						ReadyToChargeRunOutTMR_TON (IN := TRUE, PT := ReadyToChargeRunOutTMR_PT, ET=>ReadyToChargeRunOutTMR_ET);
						IF ReadyToChargeRunOutTMR_TON.Q = TRUE THEN
							Trips_DB.MachineTimedOut := TRUE;
							eMagState := E_MagState.TRIPPED;
							ReadyToChargeRunOutTMR_TON (IN := FALSE, PT := ReadyToChargeRunOutTMR_PT, ET=>ReadyToChargeRunOutTMR_ET);
						END_IF
						
						IF Permissives_DB.ChargePermOK = TRUE AND 
							MCP_IO.RemoteModeSelected = TRUE AND 
							eCommand = E_Command.CHARGE 
							THEN
								eMagState := E_MagState.CHARGING;
						ELSIF (MCP_IO.RemoteModeSelected = TRUE AND eCommand = E_Command.FULL_SHUTDOWN) 
							THEN 
								eMagState := E_MagState.FULL_SHUTDOWN;
						END_IF;
					
	//Charging State	
	E_MagState.CHARGING:	
						//send charging status to screen room
						eStatus := E_Status.CHARGING;
						
						ChargingRunOutTMR_TON (IN := TRUE, PT := ChargingRunOutTMR_PT, ET => ChargingRunOutTMR_ET);
						IF ChargingRunOutTMR_TON.Q = TRUE THEN
							Trips_DB.MachineTimedOut := TRUE;
							eMagState := E_MagState.TRIPPED;
							ChargingRunOutTMR_TON (IN := FALSE, PT := ChargingRunOutTMR_PT, ET => ChargingRunOutTMR_ET);
						END_IF
						
						IF Permissives_DB.SafetyOK THEN
						//Close all AC interlock contactor
							FOR i := 1 TO 10 BY 1 DO	
								Devices.Coil[i].CloseACInterlockRly := TRUE;
							END_FOR;
						END_IF;
	
						IF Permissives_DB.SafetyOK = TRUE AND MCP_IO.RemoteModeSelected = TRUE AND HMI_DB.StopPB = FALSE THEN
						//Close all Charge Relays
							FOR i := 1 TO 10 BY 1 DO	
								Devices.Coil[i].closeChargeRelay := TRUE;	
							END_FOR;	
						END_IF;
						
						IF Permissives_DB.AllChargerRelay_Closed = TRUE THEN
							//wait 500ms before turning on chargers
							timerBTW_ChrgRly_ChrgEnable_Chrging_TON (IN := TRUE, PT := timerBTW_ChrgRly_ChrgEnable_PT, ET => timerBTW_ChrgRly_ChrgEnable_ET);
							IF timerBTW_ChrgRly_ChrgEnable_Chrging_TON.Q = TRUE THEN 
								FOR i := 1 TO 10 BY 1 DO	
									Devices.Coil[i].enableOutputToCharger := TRUE;  //turn on all chargers	
								END_FOR;
							END_IF;	
							timerBTW_ChrgRly_ChrgEnable_Chrging_TON (IN := FALSE, PT := timerBTW_ChrgRly_ChrgEnable_PT, ET => timerBTW_ChrgRly_ChrgEnable_ET);
						ELSE 
							eMagState := E_MagState.DUMPING;
						END_IF;
	
						IF Permissives_DB.AllChargerEnabled = TRUE AND Permissives_DB.AlldcPSUok = TRUE THEN 
							//wait 10sec before setting the setpoint (Darren's sequence)
							timerForChargertoTurnOn_TON (IN := TRUE, PT := timerForChargertoTurnOn_PT, ET => timerForChargertoTurnOn_ET);
			
							IF timerForChargertoTurnOn_TON.Q = TRUE THEN
								//ChargersReady := TRUE;
								FOR i := 1 TO 10 BY 1 DO	
									Devices.Coil[i].currentSetpoint := Setpoints.Coil[i].RecipeLocal.currentSetpoint;	//setpoints from recipe	
									Devices.Coil[i].chargerSetpoint := Setpoints.Coil[i].RecipeLocal.chargerSetpoint;	//setpoints from recipe		
								END_FOR;
								timerForChargertoTurnOn_TON (IN := FALSE);
							END_IF;	
						ELSE 
							timerForChargertoTurnOn_TON (IN := FALSE);
						END_IF;
						
						// IF in manual mode and HMI pause pb is pressed | in auto mode and command from screenroom goes to pause charge, go to pause charge mode.
						IF (HMI_DB.PausePB AND MCP_IO.RemoteModeSelected = FALSE) THEN
							eMagState := E_MagState.CHARGE_PAUSED;
						END_IF;
						
						// IF in manual mode, Dump PB is pressed, go to dump mode, IF auto mode is selected, and command from screen room asks to dump go to dump mode.
						IF (HMI_DB.dumpPB = TRUE AND MCP_IO.RemoteModeSelected = FALSE) OR (MCP_IO.RemoteModeSelected = TRUE AND eCommand = E_Command.DUMP) THEN 
							eMagState := E_magState.DUMPING;
						END_IF;
						
						// if ultracap over voltage go to charge paused 
						IF Devices.Coil[i].CapWarning = TRUE THEN
							eMagState := E_MagState.CHARGE_PAUSED;
						END_IF;
						
						//IF Cap voltage = charger voltages is reached, Ready_TO_SHOOT  _ need to be recipe user input voltage
						
						IF Permissives_DB.AllCoilCapsCharged = TRUE AND GVL.AllChargerReadywithSP = TRUE
							THEN
								GVL.charge_to_readyToShoot := TRUE;
							ELSE
								GVL.charge_to_readyToShoot := FALSE;
						END_IF;
						
						IF GVL.charge_to_readyToShoot = TRUE THEN
							eMagState := E_MagState.READY_TO_SHOOT;	
							timerForChargertoTurnOn_TON (IN := FALSE, PT := timerForChargertoTurnOn_PT);
						END_IF;
		
	//Charge Paused State	
	E_MagState.CHARGE_PAUSED:
						// send status to screen room
						eStatus := E_Status.CHARGING_PAUSED;
						//Start RUNout timer
						ChargePausedRunOutTMR_TON (IN := TRUE, PT := ChargePausedRunOutTMR_PT, ET=> ChargePausedRunOutTMR_ET);// Recipe.General.ChargeRunOutTime);
						
						//Turn on disable charger
						FOR i := 1 TO 10 BY 1 DO
							Devices.Coil[i].enableOutputToCharger := FALSE;
						END_FOR;
						//wait 500ms
						timerBTW_ChrgRly_ChrgEnable_ChrgPause_TON (IN := TRUE, PT := timerBTW_ChrgEnable_ChrgRly_PT, ET => timerBTW_ChrgEnable_ChrgRly_ET);
						
						//open charger relay
						IF timerBTW_ChrgRly_ChrgEnable_ChrgPause_TON.Q = TRUE THEN
							FOR i := 1 TO 10 BY 1 DO
								Devices.Coil[i].closeChargeRelay := FALSE;
							END_FOR;
							timerBTW_ChrgRly_ChrgEnable_ChrgPause_TON (IN := FALSE, PT := timerBTW_ChrgRly_ChrgEnable_PT);
						END_IF
						IF HMI_DB.StopPB = TRUE OR (MCP_IO.RemoteModeSelected AND Permissives_DB.SafetyOK = FALSE) THEN 
							eMagState := E_MagState.DUMPING;	
						END_IF;
			
						//IF CANBus Warning/fault goes away, go back to charging
					
						IF (Devices.Coil[1].CapWarning = FALSE OR Devices.Coil[1].CoilEnabled = FALSE) AND
							(Devices.Coil[2].CapWarning = FALSE OR Devices.Coil[2].CoilEnabled = FALSE) AND
							(Devices.Coil[3].CapWarning = FALSE OR Devices.Coil[3].CoilEnabled = FALSE) AND
							(Devices.Coil[4].CapWarning = FALSE OR Devices.Coil[4].CoilEnabled = FALSE) AND
							(Devices.Coil[5].CapWarning = FALSE OR Devices.Coil[5].CoilEnabled = FALSE) AND
							(Devices.Coil[6].CapWarning = FALSE OR Devices.Coil[6].CoilEnabled = FALSE) AND
							(Devices.Coil[7].CapWarning = FALSE OR Devices.Coil[7].CoilEnabled = FALSE) AND
							(Devices.Coil[8].CapWarning = FALSE OR Devices.Coil[8].CoilEnabled = FALSE) AND
							(Devices.Coil[9].CapWarning = FALSE OR Devices.Coil[9].CoilEnabled = FALSE) AND
							(Devices.Coil[10].CapWarning = FALSE OR Devices.Coil[10].CoilEnabled = FALSE) 
						THEN
							eMagState := E_MagState.CHARGING;
						END_IF;
						
						//When RUNout timer runs out, and still in shooting state, trip the system
						IF ChargePausedRunOutTMR_TON.Q THEN
							Trips_DB.MachineTimedOut := TRUE;
							eMagState := E_MagState.TRIPPED;
							//reset timer
							ChargePausedRunOutTMR_TON (IN := FALSE, PT := ChargePausedRunOutTMR_PT, ET=> ChargePausedRunOutTMR_ET);
						END_IF;
 
						
	 E_MagState.READY_TO_SHOOT:
	 
						GVL.charge_to_readyToShoot := FALSE;
						
						//Start RUNout timer
						ReadyToShootRunOutTMR_TON (IN := TRUE, PT := ReadyToShootRunOutTMR_PT, ET => ReadyToShootRunOutTMR_ET);
						
						IF GVL.AllChargerReadywithSP = FALSE THEN
							eMagState := E_MagState.CHARGING;
						END_IF
						
						//when it is ready to shoot, disable chargers
						FOR i := 1 TO 10 BY 1 DO
							Devices.Coil[i].enableOutputToCharger := FALSE;
						END_FOR;
						//wait 500ms
						timerBTW_ChrgRly_ChrgEnable_ReadyToShoot_TON (IN := TRUE, PT := timerBTW_ChrgRly_ChrgEnable_PT, ET => timerBTW_ChrgRly_ChrgEnable_ET);
						
						//open all charger relays and AC interlock relays
						IF timerBTW_ChrgRly_ChrgEnable_ReadyToShoot_TON.Q = TRUE THEN
							FOR i := 1 TO 10 BY 1 DO
								Devices.Coil[i].closeChargeRelay := FALSE;
								Devices.Coil[i].CloseACInterlockRly := FALSE;
								//set current setpoint 
								Devices.Coil[i].currentSetpoint := Setpoints.Coil[i].RecipeLocal.currentSetpoint;
							END_FOR;
							timerBTW_ChrgRly_ChrgEnable_ReadyToShoot_TON (IN := FALSE);
						END_IF;
						
						IF Trips_DB.SystemTripped = FALSE AND Permissives_DB.ShootPermOK = TRUE THEN
							eStatus := E_Status.READY_TO_SHOOT;  //send status to screen room
							GVL.readyToShoot_to_Shoot := TRUE;
						ELSIF (Trips_DB.SystemTripped = TRUE OR Permissives_DB.ShootPermOK = FALSE OR eCommand = E_Command.DUMP) THEN
							GVL.readyToShoot_to_Shoot := FALSE;
							eMagState := E_MagState.DUMPING;
						END_IF;

						IF GVL.readyToShoot_to_Shoot = TRUE AND eCommand = E_Command.SHOOT THEN
			
							eMagState := E_MagState.SHOOTING;
						END_IF;
						
						IF MCP_IO.RemoteModeSelected = TRUE AND eCommand = E_Command.FULL_SHUTDOWN THEN
							GVL.readyToShoot_to_Shoot := FALSE;
							eMagState := E_MagState.FULL_SHUTDOWN;
						END_IF;
						
						//When RUNout timer runs out, and still in shooting state, trip the system
						IF ReadyToShootRunOutTMR_TON.Q THEN
							Trips_DB.MachineTimedOut := TRUE;
							eMagState := E_MagState.TRIPPED;
							//reset timer
							ReadyToShootRunOutTMR_TON (IN := FALSE, PT := ReadyToShootRunOutTMR_PT, ET => ReadyToShootRunOutTMR_ET);
						END_IF;
		
	E_MagState.SHOOTING:
	 					// turn off the readyToShoot_TO_Shoot bit 
						GVL.readyToShoot_to_Shoot := FALSE;
						
						//report shooting state to screen room
						eStatus := E_Status.SHOOTING;
						
						ShootingRunOutTMR_TON (IN := TRUE, PT := ShootingRunOutTMR_PT, ET => ShootingRunOutTMR_ET);
						
						FOR i := 1 TO 10 BY 1 DO
							Devices.Coil[i].CloseHVisolationRelay := TRUE;
						END_FOR;
						
						//send current feedback to screenroom, something :=  Devices.Coil[i].CurrentFeedback; ????
						
						//if screen room ask to dump, or in manual mode and stopPB or dumpPB is pressed go to dump mode
						IF eCommand = E_Command.DUMP OR (MCP_IO.RemoteModeSelected = FALSE AND (HMI_DB.dumpPB= TRUE OR HMI_DB.StopPB = TRUE)) THEN
							eMagState := E_MagState.DUMPING;
						END_IF;
						
						timerBTW_Shoot_PostShot_TON (IN := TRUE, PT := timerBTW_Shoot_PostShot_PT, ET=> timerBTW_Shoot_PostShot_ET);
				
						IF timerBTW_Shoot_PostShot_TON.Q = TRUE THEN
							GVL.shoot_to_postShot := TRUE;
							timerBTW_Shoot_PostShot_TON (IN := FALSE, PT := timerBTW_Shoot_PostShot_PT, ET=> timerBTW_Shoot_PostShot_ET);
							ELSE
								GVL.shoot_to_postShot := FALSE;
						END_IF;
						
						IF Trips_DB.SystemTripped = FALSE THEN	
							GVL.shot_going_OK := TRUE;
							ELSE
								GVL.shot_going_OK := FALSE;
						END_IF;
						
						IF GVL.shoot_to_postShot = TRUE AND GVL.shot_going_OK = TRUE THEN
							eMagState := E_MagState.POST_SHOT;
							ELSE IF ShootingRunOutTMR_TON.Q = TRUE THEN 
								Trips_DB.MachineTimedOut := TRUE;
								eMagState := E_MagState.TRIPPED;
								ShootingRunOutTMR_TON (IN := FALSE, PT := ShootingRunOutTMR_PT, ET => ShootingRunOutTMR_ET);
							END_IF
						END_IF;		
		
	E_MagState.POST_SHOT:
						GVL.shoot_to_postShot := FALSE;
						
						PostShotRunOutTMR_TON (IN := TRUE, PT := PostShotRunOutTMR_PT, ET => PostShotRunOutTMR_ET);
						
						//Send status to screenroom
						eStatus := E_Status.POST_SHOT;
						//open HV isolation Relays
						FOR i := 1 TO 10 BY 1 DO
							Devices.Coil[i].CloseHVisolationRelay := FALSE;
						END_FOR;
						
						//if temperature are all good and safety is okay, shot is done
						IF Permissives_DB.SafetyOK = TRUE AND Devices.Coil[i].ChargeVoltageFeedback <= 10 THEN
							GVL.shot_is_done := TRUE;
							ELSE
								GVL.shot_is_done := FALSE;
						END_IF;
						
						//if shot is done, go back to idle state  // it was shot is done or command.idle
						IF GVL.shot_is_done = TRUE AND (MCP_IO.RemoteModeSelected = TRUE AND eCommand = E_Command.IDLE) THEN
							eMagState := E_MagState.IDLE;
						//if screen room ask to dump, or in manual mode and stopPB or dumpPB is pressed go to dump mode
						ELSIF eCommand = E_Command.DUMP OR (MCP_IO.RemoteModeSelected = FALSE AND (HMI_DB.dumpPB= TRUE OR HMI_DB.StopPB = TRUE)) THEN
							eMagState := E_MagState.DUMPING;
						ELSIF (MCP_IO.RemoteModeSelected = TRUE AND eCommand = E_Command.FULL_SHUTDOWN) THEN 
							eMagState := E_MagState.FULL_SHUTDOWN;
						END_IF;
						
						IF PostShotRunOutTMR_TON.Q = TRUE THEN
							Trips_DB.MachineTimedOut := TRUE;
							eMagState := E_MagState.TRIPPED;
							PostShotRunOutTMR_TON (IN := FALSE, PT := PostShotRunOutTMR_PT, ET => PostShotRunOutTMR_ET);
						END_IF
								
	E_MagState.DUMPING:	
						//disable all chargers
						FOR i := 1 TO 10 BY 1 DO
							Devices.Coil[i].enableOutputToCharger := FALSE;
							Devices.Coil[i].CloseHVisolationRelay := FALSE;   //Open all HV isolation relays
						END_FOR
						
						IF Permissives_DB.AllChargerEnabled = FALSE THEN 
							timerBTW_ChrgEnable_ChrgRly_Dumping_TON (IN := TRUE, PT := timerBTW_ChrgRly_ChrgEnable_PT, ET=>timerBTW_ChrgEnable_ChrgRly_Dumping_ET); 					 
						ELSE
							timerBTW_ChrgEnable_ChrgRly_Dumping_TON (IN := FALSE);
						END_IF;
						
						IF timerBTW_ChrgEnable_ChrgRly_Dumping_TON.Q = TRUE THEN
							FOR i := 1 TO 10 BY 1 DO
								Devices.Coil[i].closeChargeRelay := FALSE; //open charge relay
							END_FOR;
							timerBTW_ChrgEnable_ChrgRly_Dumping_TON (IN := FALSE);
						END_IF;
						
						//Close all dump relays
						Devices.Coil[1].OpenDumpRelays := FALSE; //NC so close dump relays
						Devices.Coil[2].OpenDumpRelays := FALSE;
						Devices.Coil[3].OpenDumpRelays := FALSE;
						Devices.Coil[4].OpenDumpRelays := FALSE;
						Devices.Coil[5].OpenDumpRelays := FALSE;
						Devices.Coil[6].OpenDumpRelays := FALSE;
						Devices.Coil[7].OpenDumpRelays := FALSE;
						Devices.Coil[8].OpenDumpRelays := FALSE;
						Devices.Coil[9].OpenDumpRelays := FALSE;
						Devices.Coil[10].OpenDumpRelays := FALSE;
						
						//send state to screen room
						eStatus := E_Status.DUMPING;
						
						DumpingRunOutTMR_TON (IN := TRUE, PT := DumpingRunOutTMR_PT, ET => DumpingRunOutTMR_ET);
						IF DumpingRunOutTMR_TON.Q = TRUE THEN
							Trips_DB.MachineTimedOut := TRUE;
							eMagState := E_MagState.TRIPPED;
							DumpingRunOutTMR_TON (IN := FALSE, PT := DumpingRunOutTMR_PT, ET => DumpingRunOutTMR_ET);
						END_IF
						
						//NC, if all dump relays are closed, and all cap voltage discharged, start timer and go back to IDLE automaticlally
						IF Permissives_DB.AllDumpRelayOpen = FALSE AND Permissives_DB.AllCoilCapsCharged = FALSE THEN 
							timerBTW_DUMP_IDLE (IN := TRUE, PT := timerBTW_DUMP_IDLE_PT, ET => timerBTW_DUMP_IDLE_ET);
							IF timerBTW_DUMP_IDLE.Q = TRUE THEN 
								GVL.dump_to_idle := TRUE;
							END_IF;	
						ELSE
							timerBTW_DUMP_IDLE (IN := FALSE);
							GVL.dump_to_idle := FALSE;	
						END_IF;
						
						IF GVL.dump_to_idle = TRUE THEN
							eMagState := E_MagState.IDLE;
							timerBTW_DUMP_IDLE (IN := FALSE, PT := timerBTW_DUMP_IDLE_PT);
						ELSIF GVL.dump_to_idle = TRUE AND MCP_IO.RemoteModeSelected = TRUE AND eCommand = E_Command.FULL_SHUTDOWN THEN
								eMagState := E_MagState.FULL_SHUTDOWN;
						END_IF;
						//GVL.dump_to_idle := FALSE;
						
	E_MagState.TRIPPED: 
						eStatus := E_Status.TRIPPED;	
						
						FOR i := 1 TO 10 BY 1 DO
							//Disable all Chargers
							Devices.Coil[i].enableOutputToCharger := FALSE;
		
							//open (de-energize) all interlock relays
							Devices.Coil[i].CloseACInterlockRly := FALSE;
	
							//Close (de-energize) All Dump relays
							Devices.Coil[i].OpenDumpRelays := FALSE;
							
							Devices.Coil[i].CloseHVisolationRelay := FALSE;   //Open all HV isolation relays
						END_FOR;
						//wait 500ms before opening the charge relay
						timerBTW_ChrgEnable_ChrgRly_Tripped_TON (IN := TRUE, PT := timerBTW_ChrgEnable_ChrgRly_PT, ET => timerBTW_ChrgEnable_ChrgRly_Tripped_ET);
						
						IF timerBTW_ChrgEnable_ChrgRly_Tripped_TON.Q = TRUE THEN
							FOR i := 1 TO 10 BY 1 DO
							//open all charge relays
							Devices.Coil[i].closeChargeRelay := FALSE;
							END_FOR;
							timerBTW_ChrgEnable_ChrgRly_Tripped_TON (IN := FALSE, PT := timerBTW_ChrgEnable_ChrgRly_PT, ET => timerBTW_ChrgEnable_ChrgRly_Tripped_ET);
						END_IF;
						
						// when Trip is clear by the opeartor, it goes back to idle state.
						IF Trips_DB.SystemTripped = FALSE AND Permissives_DB.SafetyOK = TRUE THEN 
							eMagState := E_MagState.IDLE;
						END_IF;
						
						//reset all run out tmr
						ReadyToChargeRunOutTMR_TON (IN := FALSE, PT := ReadyToChargeRunOutTMR_PT, ET=>ReadyToChargeRunOutTMR_ET);
						ChargingRunOutTMR_TON (IN := FALSE, PT := ChargingRunOutTMR_PT, ET => ChargingRunOutTMR_ET);
						ChargePausedRunOutTMR_TON (IN := FALSE, PT := ChargePausedRunOutTMR_PT, ET=> ChargePausedRunOutTMR_ET);
						ReadyToShootRunOutTMR_TON (IN := FALSE, PT := ReadyToShootRunOutTMR_PT, ET => ReadyToShootRunOutTMR_ET);
						ShootingRunOutTMR_TON (IN := FALSE, PT := ShootingRunOutTMR_PT, ET => ShootingRunOutTMR_ET);
						PostShotRunOutTMR_TON (IN := FALSE, PT := PostShotRunOutTMR_PT, ET => PostShotRunOutTMR_ET);
						DumpingRunOutTMR_TON (IN := FALSE, PT := DumpingRunOutTMR_PT, ET => DumpingRunOutTMR_ET);
						
END_CASE

//run hmi 
HMI();

//reset counter
IF i > 10 THEN 
	i := 1;
END_IF;

END_PROGRAM

// ---- POUs/MAIN.TcPOU
PROGRAM MAIN
VAR
	
	status0:BOOL;
	
END_VAR

Alias();
CAN_comm();
Tx_MasterPLC();
AnalogConversion();
//Permissives();
//Trips();
MODE_SELECTION_1();
//Alarms();
Heartbeat();
VoltageOutputCal();
//Cal_ChargeTime();


//test
//IF MCP_IO.AutoModeSelected THEN
//	Output.R2_05_07 := heartbeat.pulse_1Hz;
//END_IF

	
//sample test
IF gvl.test = TRUE THEN
	Output.R2_05_00 := TRUE;
	ELSE 
		Output.R2_05_00 := FALSE; 	
END_IF;

END_PROGRAM

// ---- POUs/VoltageOutputCal.TcPOU
PROGRAM VoltageOutputCal
VAR
	i : INT := 1;
END_VAR

// charger setpoint = (num of caps * x - ax + bY)/ time;
Devices.Coil[i].chargerSetpoint := Setpoints.Coil[i].RecipeLocal.chargerSetpoint; //charger setpoint voltage is calculated from the recipe current and num of caps.

//

FOR i := 1 TO 10 BY 1 DO
	//set current setpoint 
	Setpoints.Coil[i].RecipeLocal.currentSetpoint := REAL_TO_INT (Recipe.Coil[i].currentSetpoint);
	//Setpoints.Coil[i].RecipeLocal.chargerSetpoint := REAL_TO_INT (Recipe.Coil[i].chargerSetpoint);
	Setpoints.Coil[i].Recipe.CoilEnable := Recipe.Coil[i].CoilEnable;
	Setpoints.Coil[i].RecipeLocal.CurrentDuration := REAL_TO_TIME (Recipe.Coil[i].CurrentDuration*1000);
	
	//total voltage
	Devices.Coil[i].TotalVoltage := Devices.Coil[i].CapVoltage[1]+
									Devices.Coil[i].CapVoltage[2]+
									Devices.Coil[i].CapVoltage[3]+
									Devices.Coil[i].CapVoltage[4]+
									Devices.Coil[i].CapVoltage[5]+
									Devices.Coil[i].CapVoltage[6]+
									Devices.Coil[i].CapVoltage[7]+
									Devices.Coil[i].CapVoltage[8]+
									Devices.Coil[i].CapVoltage[9]+
									Devices.Coil[i].CapVoltage[10]+
									Devices.Coil[i].CapVoltage[11]+
									Devices.Coil[i].CapVoltage[12]+
									Devices.Coil[i].CapVoltage[13]+
									Devices.Coil[i].CapVoltage[14]+
									Devices.Coil[i].CapVoltage[15];
END_FOR;


IF i > 10 THEN 
	i := 1;
END_IF

END_PROGRAM

// ---- POUs/Permissives.TcPOU
PROGRAM Permissives
VAR

	stPermissives			: ST_PermissivesToMainPLC;
	
	AdminFaultBypassOn		: BOOL;
	
	i : INT := 1;
	j : INT := 1;	
END_VAR

//HMI Admin bypass button
AdminFaultBypassOn := HMI_DB.SafetyOK;

//Check to see if any coil is disabled
IF Devices.Coil[1].CoilEnabled = FALSE OR
	Devices.Coil[2].CoilEnabled = FALSE OR
	Devices.Coil[3].CoilEnabled = FALSE OR
	Devices.Coil[4].CoilEnabled = FALSE OR
	Devices.Coil[5].CoilEnabled = FALSE OR
	Devices.Coil[6].CoilEnabled = FALSE OR
	Devices.Coil[7].CoilEnabled = FALSE OR
	Devices.Coil[8].CoilEnabled = FALSE OR
	Devices.Coil[9].CoilEnabled = FALSE OR
	Devices.Coil[10].CoilEnabled = FALSE 
	THEN
		Permissives_DB.AnyCoilDisabled := TRUE;
	ELSE
		Permissives_DB.AnyCoilDisabled := FALSE;
END_IF;

//check to see if each LCP system is ready based on the selected safety parameters.
FOR i := 1 TO 10 BY 1 DO
	IF Devices.Coil[i].AC_Interlock_RlyClose = TRUE AND 
		Devices.Coil[i].ChargeRelay_closed = TRUE AND
		Devices.Coil[i].CoilTemperatureHigh = FALSE AND
		Devices.Coil[i].DumpResistorTemperatureHigh = FALSE AND
		Devices.Coil[i].DumpRelay1_closed = TRUE AND
		Devices.Coil[i].DumpRelay2_closed = TRUE AND
		Devices.Coil[i].FlybackD1_Alive = TRUE AND
		Devices.Coil[i].FlybackD2_Alive = TRUE AND
		Devices.Coil[i].GroundLoopCurrentDetected = FALSE AND
		Devices.Coil[i].Local_StopPB_Pressed = FALSE AND
		Devices.Coil[i].LossPneumaticPressure = FALSE 
		THEN
			Devices.Coil[i].SystemReady := TRUE;
		ELSE
			Devices.Coil[i].SystemReady := FALSE;
	END_IF;
END_FOR;


//Safety Permissives
	//Interlock Safety
	IF (Devices.Coil[1].AC_Interlock_RlyClose = TRUE OR Devices.Coil[1].CoilEnabled = FALSE) AND 
		(Devices.Coil[2].AC_Interlock_RlyClose = TRUE OR Devices.Coil[2].CoilEnabled = FALSE) AND 
		(Devices.Coil[3].AC_Interlock_RlyClose = TRUE OR Devices.Coil[3].CoilEnabled = FALSE) AND
		(Devices.Coil[4].AC_Interlock_RlyClose = TRUE OR Devices.Coil[4].CoilEnabled = FALSE) AND
		(Devices.Coil[5].AC_Interlock_RlyClose = TRUE OR Devices.Coil[5].CoilEnabled = FALSE) AND
		(Devices.Coil[6].AC_Interlock_RlyClose = TRUE OR Devices.Coil[6].CoilEnabled = FALSE) AND
		(Devices.Coil[7].AC_Interlock_RlyClose = TRUE OR Devices.Coil[7].CoilEnabled = FALSE) AND
		(Devices.Coil[8].AC_Interlock_RlyClose = TRUE OR Devices.Coil[8].CoilEnabled = FALSE) AND
		(Devices.Coil[9].AC_Interlock_RlyClose = TRUE OR Devices.Coil[9].CoilEnabled = FALSE) AND 
		(Devices.Coil[10].AC_Interlock_RlyClose = TRUE OR Devices.Coil[10].CoilEnabled = FALSE)
		
		THEN 
			Permissives_DB.AllacInterlock_Closed := TRUE;
		ELSE 
			Permissives_DB.AllacInterlock_Closed := FALSE;
	END_IF;

	//Coil Temperature
	IF Devices.Coil[1].CoilTemperatureHigh = FALSE AND
		Devices.Coil[2].CoilTemperatureHigh = FALSE 
		THEN
			Permissives_DB.All_Coil_TemperatureOK := TRUE;
		ELSE 
			Permissives_DB.All_Coil_TemperatureOK := FALSE;
	END_IF;

	//Dump Resistor Temperature
	IF Devices.Coil[1].DumpResistorTemperatureHigh = FALSE AND
		Devices.Coil[2].DumpResistorTemperatureHigh = FALSE 
		THEN
			Permissives_DB.AllDumpResistorTempOK := TRUE;
		ELSE 
			Permissives_DB.AllDumpResistorTempOK := FALSE;
	END_IF;
	
	//Ground loop current
	IF Devices.Coil[1].GroundLoopCurrentDetected = FALSE AND
		Devices.Coil[2].GroundLoopCurrentDetected = FALSE 
		THEN
			Permissives_DB.NoGroundLoopCurrentDetected := TRUE;
		ELSE 
			Permissives_DB.NoGroundLoopCurrentDetected := FALSE;
	END_IF;
	
	//Flyback Diodes - Not enought time for PI3 - temporarily disabled for PI3
(*	IF ((Devices.coil[1].FlybackD1_Alive = TRUE AND Devices.coil[1].FlybackD2_Alive = TRUE) OR Devices.Coil[1].CoilEnabled = FALSE) AND
		((Devices.coil[2].FlybackD1_Alive = TRUE AND Devices.coil[2].FlybackD2_Alive = TRUE) OR Devices.Coil[2].CoilEnabled = FALSE)
		THEN 
			AllFlybackDiodes_Alive := TRUE;
		ELSE 
			AllFlybackDiodes_Alive := FALSE;
	END_IF;
*)	
	IF (Permissives_DB.All_Coil_TemperatureOK = TRUE AND
		Permissives_DB.AllDumpResistorTempOK = TRUE AND
		Permissives_DB.NoGroundLoopCurrentDetected = TRUE AND
		//AllFlybackDiodes_Alive = TRUE AND 
		Trips_DB.AnyACInterlockFail = FALSE AND
		Trips_DB.AnyHVisoRelayFailed = FALSE AND
		Trips_DB.AnyChargeRlyFail = FALSE AND
		Trips_DB.AnyDumpRlyFail = FALSE AND
		Trips_DB.AnyEstopPressed = FALSE AND
		Permissives_DB.AlldcPSUok = TRUE AND
		MCP_IO.CageEstopCircuitOK = TRUE) OR HMI_DB.SafetyOK = TRUE 
		THEN
			Permissives_DB.SafetyOK := TRUE;
		ELSE 
			Permissives_DB.SafetyOK := FALSE; 
	END_IF;

//Charger Active Status - obsolete
(*
IF (Devices.Coil[1].PSU0_active = TRUE OR Devices.Coil[1].CoilEnabled = FALSE) AND
	(Devices.Coil[2].PSU0_active = TRUE OR Devices.Coil[2].CoilEnabled = FALSE) //AND
	//Coil3.PSU.active AND 
	THEN 
		AllChargers_Active := TRUE;
	ELSE 
		AllChargers_Active := FALSE;
END_IF;
*)

IF (Devices.Coil[1].PSU1_DCOK = TRUE OR Devices.Coil[1].CoilEnabled = FALSE) AND
	(Devices.Coil[2].PSU1_DCOK = TRUE OR Devices.Coil[2].CoilEnabled = FALSE) (*AND Coil3.PSU.active*) AND
	MCP_IO.PSU1_DCOK = TRUE
	THEN 
		Permissives_DB.AlldcPSUok := TRUE;
	ELSE 
		Permissives_DB.AlldcPSUok := FALSE;
END_IF;

//Charger Enabled Status
IF (Devices.Coil[1].ChargerIsEnabled = TRUE OR Devices.Coil[1].CoilEnabled = FALSE) AND
	(Devices.Coil[2].ChargerIsEnabled = TRUE OR Devices.Coil[2].CoilEnabled = FALSE) AND
	(Devices.Coil[3].ChargerIsEnabled = TRUE OR Devices.Coil[3].CoilEnabled = FALSE) AND
	(Devices.Coil[4].ChargerIsEnabled = TRUE OR Devices.Coil[4].CoilEnabled = FALSE) AND
	(Devices.Coil[5].ChargerIsEnabled = TRUE OR Devices.Coil[5].CoilEnabled = FALSE) AND
	(Devices.Coil[6].ChargerIsEnabled = TRUE OR Devices.Coil[6].CoilEnabled = FALSE) AND
	(Devices.Coil[7].ChargerIsEnabled = TRUE OR Devices.Coil[7].CoilEnabled = FALSE) AND	
	(Devices.Coil[8].ChargerIsEnabled = TRUE OR Devices.Coil[8].CoilEnabled = FALSE) AND
	(Devices.Coil[9].ChargerIsEnabled = TRUE OR Devices.Coil[9].CoilEnabled = FALSE) AND
	(Devices.Coil[10].ChargerIsEnabled = TRUE OR Devices.Coil[10].CoilEnabled = FALSE) 
	THEN 
		Permissives_DB.AllChargerEnabled := TRUE;
	ELSE 
		Permissives_DB.AllChargerEnabled := FALSE;
END_IF

//???? need more work
IF ((Devices.Coil[1].chargerSetpoint >= Setpoints.Coil[1].RecipeLocal.chargerSetpoint) OR Devices.Coil[1].CoilEnabled = FALSE) AND
	((Devices.Coil[2].chargerSetpoint >= Setpoints.Coil[2].RecipeLocal.chargerSetpoint) OR Devices.Coil[2].CoilEnabled = FALSE) AND 
	((Devices.Coil[3].chargerSetpoint >= Setpoints.Coil[3].RecipeLocal.chargerSetpoint) OR Devices.Coil[3].CoilEnabled = FALSE) AND
	((Devices.Coil[4].chargerSetpoint >= Setpoints.Coil[4].RecipeLocal.chargerSetpoint) OR Devices.Coil[4].CoilEnabled = FALSE) AND
	((Devices.Coil[5].chargerSetpoint >= Setpoints.Coil[5].RecipeLocal.chargerSetpoint) OR Devices.Coil[5].CoilEnabled = FALSE) AND
	((Devices.Coil[6].chargerSetpoint >= Setpoints.Coil[6].RecipeLocal.chargerSetpoint) OR Devices.Coil[6].CoilEnabled = FALSE) AND
	((Devices.Coil[7].chargerSetpoint >= Setpoints.Coil[7].RecipeLocal.chargerSetpoint) OR Devices.Coil[7].CoilEnabled = FALSE) AND
	((Devices.Coil[8].chargerSetpoint >= Setpoints.Coil[8].RecipeLocal.chargerSetpoint) OR Devices.Coil[8].CoilEnabled = FALSE) AND
	((Devices.Coil[9].chargerSetpoint >= Setpoints.Coil[9].RecipeLocal.chargerSetpoint) OR Devices.Coil[9].CoilEnabled = FALSE) AND
	((Devices.Coil[10].chargerSetpoint >= Setpoints.Coil[10].RecipeLocal.chargerSetpoint) OR Devices.Coil[10].CoilEnabled = FALSE)
	THEN
		GVL.AllChargerReadywithSP := TRUE;
	ELSE
		GVL.AllChargerReadywithSP := FALSE;
END_IF;

//check to see if all cap voltage ready to shoot
FOR i := 1 TO 10 BY 1 DO
		IF ((Devices.Coil[i].CapVoltage[1] >= Devices.Coil[i].chargerSetpoint) AND
			(Devices.Coil[i].CapVoltage[2] >= Devices.Coil[i].chargerSetpoint) AND
			(Devices.Coil[i].CapVoltage[3] >= Devices.Coil[i].chargerSetpoint) AND
			(Devices.Coil[i].CapVoltage[4] >= Devices.Coil[i].chargerSetpoint) AND
			(Devices.Coil[i].CapVoltage[5] >= Devices.Coil[i].chargerSetpoint) AND
			(Devices.Coil[i].CapVoltage[6] >= Devices.Coil[i].chargerSetpoint) AND
			(Devices.Coil[i].CapVoltage[7] >= Devices.Coil[i].chargerSetpoint) AND
			(Devices.Coil[i].CapVoltage[8] >= Devices.Coil[i].chargerSetpoint) AND
			(Devices.Coil[i].CapVoltage[9] >= Devices.Coil[i].chargerSetpoint) AND
			(Devices.Coil[i].CapVoltage[10] >= Devices.Coil[i].chargerSetpoint)) OR 
			Devices.Coil[i].CoilEnabled = FALSE
		THEN
			Devices.Coil[i].AllCapsCharged := TRUE;
	END_IF
END_FOR;
//check to see if all coils are charged
IF Devices.Coil[1].AllCapsCharged = TRUE AND 
	Devices.Coil[2].AllCapsCharged = TRUE AND 
	Devices.Coil[3].AllCapsCharged = TRUE AND 
	Devices.Coil[4].AllCapsCharged = TRUE AND 
	Devices.Coil[5].AllCapsCharged = TRUE AND 
	Devices.Coil[6].AllCapsCharged = TRUE AND 
	Devices.Coil[7].AllCapsCharged = TRUE AND 
	Devices.Coil[8].AllCapsCharged = TRUE AND 
	Devices.Coil[9].AllCapsCharged = TRUE AND 
	Devices.Coil[10].AllCapsCharged = TRUE 
THEN 
	Permissives_DB.AllCoilCapsCharged := TRUE;
ELSE
	Permissives_DB.AllCoilCapsCharged := FALSE;	
END_IF

//check to see if all cap voltage drops to 1
IF ((Devices.Coil[i].CapVoltage[1] <= 1) AND
	(Devices.Coil[i].CapVoltage[2] <= 1) AND
	(Devices.Coil[i].CapVoltage[3] <= 1) AND
	(Devices.Coil[i].CapVoltage[4] <= 1) AND
	(Devices.Coil[i].CapVoltage[5] <= 1) AND
	(Devices.Coil[i].CapVoltage[6] <= 1) AND
	(Devices.Coil[i].CapVoltage[7] <= 1) AND
	(Devices.Coil[i].CapVoltage[8] <= 1) AND
	(Devices.Coil[i].CapVoltage[9] <= 1) AND
	(Devices.Coil[i].CapVoltage[10] <= 1)) OR 
	Devices.Coil[i].CoilEnabled = FALSE
THEN
	Devices.Coil[i].AllCapsCharged := FALSE;
END_IF;



//Charger Relay
IF Devices.Coil[1].ChargeRelay_closed = FALSE AND
	Devices.Coil[2].ChargeRelay_closed = FALSE 
	//coil n
	THEN
		Permissives_DB.AllChargerRelay_Closed := TRUE;
	ELSE 
		Permissives_DB.AllChargerRelay_Closed := FALSE;
END_IF

	
//Dump Relay Status
(* obsolete - use the one at the bottom
IF ((Devices.Coil[1].DumpRelay1_closed = FALSE AND Devices.Coil[1].DumpRelay2_closed = FALSE) OR Devices.Coil[1].CoilEnabled = FALSE) AND
	((Devices.Coil[2].DumpRelay1_closed = FALSE AND Devices.Coil[2].DumpRelay2_closed = FALSE) OR Devices.Coil[2].CoilEnabled = FALSE) AND
	((Devices.Coil[3].DumpRelay1_closed = FALSE AND Devices.Coil[3].DumpRelay2_closed = FALSE) OR Devices.Coil[3].CoilEnabled = FALSE) AND
	((Devices.Coil[4].DumpRelay1_closed = FALSE AND Devices.Coil[4].DumpRelay2_closed = FALSE) OR Devices.Coil[4].CoilEnabled = FALSE) AND
	((Devices.Coil[5].DumpRelay1_closed = FALSE AND Devices.Coil[5].DumpRelay2_closed = FALSE) OR Devices.Coil[5].CoilEnabled = FALSE) AND
	((Devices.Coil[6].DumpRelay1_closed = FALSE AND Devices.Coil[6].DumpRelay2_closed = FALSE) OR Devices.Coil[6].CoilEnabled = FALSE) AND
	((Devices.Coil[7].DumpRelay1_closed = FALSE AND Devices.Coil[7].DumpRelay2_closed = FALSE) OR Devices.Coil[7].CoilEnabled = FALSE) AND
	((Devices.Coil[8].DumpRelay1_closed = FALSE AND Devices.Coil[8].DumpRelay2_closed = FALSE) OR Devices.Coil[8].CoilEnabled = FALSE) AND
	((Devices.Coil[9].DumpRelay1_closed = FALSE AND Devices.Coil[9].DumpRelay2_closed = FALSE) OR Devices.Coil[9].CoilEnabled = FALSE) AND
	((Devices.Coil[10].DumpRelay1_closed = FALSE AND Devices.Coil[10].DumpRelay2_closed = FALSE) OR Devices.Coil[10].CoilEnabled = FALSE)

	THEN
		AllDumpRelayOpen := TRUE;
		ELSE 
			AllDumpRelayOpen := FALSE;
END_IF;
*)	
IF ((Devices.Coil[1].DumpRelay1_closed = TRUE AND Devices.Coil[1].DumpRelay2_closed = TRUE) OR Devices.Coil[1].CoilEnabled = FALSE) AND
	((Devices.Coil[2].DumpRelay1_closed = TRUE AND Devices.Coil[2].DumpRelay2_closed = TRUE) OR Devices.Coil[2].CoilEnabled = FALSE) AND
	((Devices.Coil[3].DumpRelay1_closed = TRUE AND Devices.Coil[3].DumpRelay2_closed = TRUE) OR Devices.Coil[3].CoilEnabled = FALSE) AND
	((Devices.Coil[4].DumpRelay1_closed = TRUE AND Devices.Coil[4].DumpRelay2_closed = TRUE) OR Devices.Coil[4].CoilEnabled = FALSE) AND
	((Devices.Coil[5].DumpRelay1_closed = TRUE AND Devices.Coil[5].DumpRelay2_closed = TRUE) OR Devices.Coil[5].CoilEnabled = FALSE) AND
	((Devices.Coil[6].DumpRelay1_closed = TRUE AND Devices.Coil[6].DumpRelay2_closed = TRUE) OR Devices.Coil[6].CoilEnabled = FALSE) AND
	((Devices.Coil[7].DumpRelay1_closed = TRUE AND Devices.Coil[7].DumpRelay2_closed = TRUE) OR Devices.Coil[7].CoilEnabled = FALSE) AND
	((Devices.Coil[8].DumpRelay1_closed = TRUE AND Devices.Coil[8].DumpRelay2_closed = TRUE) OR Devices.Coil[8].CoilEnabled = FALSE) AND
	((Devices.Coil[9].DumpRelay1_closed = TRUE AND Devices.Coil[9].DumpRelay2_closed = TRUE) OR Devices.Coil[9].CoilEnabled = FALSE) AND
	((Devices.Coil[10].DumpRelay1_closed = TRUE AND Devices.Coil[10].DumpRelay2_closed = TRUE) OR Devices.Coil[10].CoilEnabled = FALSE) 
	THEN
		Permissives_DB.AllDumpRelayOpen := FALSE;
		ELSE
			Permissives_DB.AllDumpRelayOpen := TRUE;;
END_IF;

//any pneumatic pressure loss
FOR i := 1 TO 10 BY 1 DO
	IF Devices.Coil[i].LossPneumaticPressure = FALSE THEN
		Permissives_DB.NoPneumaticPressureLoss := TRUE;
		ELSE 
			Permissives_DB.NoPneumaticPressureLoss := FALSE;
	END_IF
END_FOR

//When disable a coil, ignore the permissives of it
IF Permissives_DB.AnyCoilDisabled = TRUE THEN
	FOR i := 1 TO 10 BY 1 DO
		IF Devices.Coil[i].CoilEnabled = FALSE THEN
			Devices.Coil[i].SystemReady := TRUE;
			Devices.Coil[i].PSU0_active := TRUE;
			Devices.Coil[i].Local_StopPB_Pressed := FALSE;
			Devices.Coil[i].FlybackD1_Alive := TRUE;
			Devices.Coil[i].FlybackD2_Alive := TRUE;
			Devices.Coil[i].DumpResistorTemperatureHigh := FALSE;
			Devices.Coil[i].GroundLoopCurrentDetected := FALSE;
			Devices.Coil[i].CoilTemperatureHigh := FALSE;
			Devices.Coil[i].LossPneumaticPressure := FALSE;
			ELSE
				Devices.Coil[i].SystemReady := FALSE;
		END_IF;
	END_FOR;
END_IF;	


//TURN OFF the outputs of the coil when it is disabled
IF Permissives_DB.AnyCoilDisabled = TRUE THEN
	FOR i := 1 TO 10 BY 1 DO
		IF Devices.Coil[i].CoilEnabled = TRUE THEN
			Devices.Coil[i].CloseACInterlockRly := FALSE;
			Devices.Coil[i].OpenDumpRelays := FALSE;
			Devices.Coil[i].closeChargeRelay := FALSE;
		END_IF;
	END_FOR;
END_IF;

//*******************************************************************//	
//Charge Permissives
IF (Permissives_DB.SafetyOK = TRUE OR HMI_DB.SafetyOK) AND (Permissives_DB.AllDumpRelayOpen = TRUE OR HMI_DB.AllDumpRelaysOpen  = TRUE) AND (Trips_DB.InstrumentationFaulted = FALSE OR HMI_DB.IntrumentationFaulted = FALSE) THEN 
	Permissives_DB.ChargePermOK := TRUE;	
	ELSE Permissives_DB.ChargePermOK := FALSE;	
END_IF;


//Shoot Permissives
IF Permissives_DB.SafetyOK = TRUE AND (Permissives_DB.AlldcPSUok = FALSE OR HMI_DB.AllChargesAreActive = FALSE) AND (Permissives_DB.AllDumpRelayOpen = TRUE OR HMI_DB.AllDumpRelaysOpen = TRUE) THEN
	Permissives_DB.ShootPermOK := TRUE;
	ELSE Permissives_DB.ShootPermOK := FALSE;
END_IF;

//sending permissives to Main PLC (screen room)
stPermissives.All_Coil_TemperatureOK := Permissives_DB.All_Coil_TemperatureOK;
stPermissives.AllacInterlock_Closed := Permissives_DB.AllacInterlock_Closed;
stPermissives.AllChargerEnabled := Permissives_DB.AllChargerEnabled;
stPermissives.AllChargerRelay_Closed := Permissives_DB.AllChargerRelay_Closed;
stPermissives.AlldcPSUok := Permissives_DB.AlldcPSUok;
stPermissives.AllDumpRelayOpen := Permissives_DB.AllDumpRelayOpen;
stPermissives.AllDumpResistorTempOK := Permissives_DB.AllDumpResistorTempOK;
//stPermissives.AllFlybackDiodes_Alive := AllFylbackDiodes_Alive;
stPermissives.AnyCoilDisabled := Permissives_DB.AnyCoilDisabled;
stPermissives.ChargePermOK := Permissives_DB.ChargePermOK;
stPermissives.NoGroundLoopCurrentDetected := Permissives_DB.NoGroundLoopCurrentDetected;
stPermissives.SafetyOK := Permissives_DB.SafetyOK;
stPermissives.ShootPermOK := Permissives_DB.ShootPermOK;
stPermissives.AdminFaultBypassOn := AdminFaultBypassOn;


IF i > 10 THEN
	i := 1;
END_IF;

IF j > 10 THEN
	j := 1;
END_IF;

END_PROGRAM

// ---- POUs/Trips.TcPOU
PROGRAM Trips
VAR
	bTest							: BOOL;
	//delay2s : Delay2s;
	evtLogger						: FB_TcEventLogger;
	
	ACintLockRlyFaultDelay_PT		: TIME := T#2S;
	HVisoRlyFaultDelay_PT			: TIME := T#2S;
	DumpRly1FaultDelay_PT			: TIME := T#2S;
	//DumpRly2FaultDelay_PT			: TIME := T#2S;
	ChrgRlyFaultDelay_PT			: TIME := T#2S;
	stControl						: ST_Control;
	
	i : INT := 1; //coil num 1-10
	j : INT := 1; //cap num 1-10 or 15
END_VAR

//AI channel reading faults.

//******************** Coil 1 - Charger Voltage Instrument Fault
IF InstrumentReading.R2_01_CH00 <= 0.0 THEN
	Devices.Coil[1].ChargerVoltageFault_TON (IN := TRUE, PT := T#2S);
	Trips_DB.Coil[1].chargerVoltageReadingFaulted := Devices.Coil[1].ChargerVoltageFault_TON.Q;
ELSE 
	Devices.Coil[1].ChargerVoltageFault_TON (IN := FALSE);
	Trips_DB.Coil[1].chargerVoltageReadingFaulted := FALSE;
END_IF;


//Coil1.currentFeedback := SEL(bTest, Coil1.currentFeedback, 200);  

//********************Coil 1 - Current Instrument Fault
IF InstrumentReading.R2_01_CH01 <= 0.0 THEN
	Devices.Coil[1].CurrentSensorFault_TON (IN := TRUE, PT := T#2S);
	Trips_DB.Coil[1].CurrentReadingFaulted := Devices.Coil[1].CurrentSensorFault_TON.Q;
ELSE 
	Devices.Coil[1].CurrentSensorFault_TON (IN := FALSE);
	Trips_DB.Coil[1].CurrentReadingFaulted := FALSE;
END_IF


//********************Coil 1 - B-field Instrument Fault  --  this one is a good one.
(*
IF InstrumentReading.R2_01_CH02 <= 0.0 THEN
	Devices.Coil[1].BfieldSensorFault_TON (IN := TRUE, PT := T#2S);
	Trips_DB.Coil1_BfieldReadingFaulted := Devices.Coil[1].BfieldSensorFault_TON.Q;
ELSE 
	Devices.Coil[1].BfieldSensorFault_TON (IN := FALSE);
	Trips_DB.Coil1_BfieldReadingFaulted := FALSE;   
END_IF
*)

//Instrumentation Faults
FOR i := 1 TO 10 BY 1 DO
	IF Trips_DB.Coil[i].ChargerVoltageReadingFaulted = TRUE //OR
		//Trips_DB.Coil[i].currentReadingFaulted = TRUE OR  //-- commented out for PI3
		//Trips_DB.Coil[i].BfieldReadingFaulted = TRUE
		THEN
			Trips_DB.InstrumentationFaulted := TRUE;
	END_IF;
END_FOR;

//********************Relay fail to close Trips
FOR i := 1 TO 10 BY 1 DO
	//check to see if AC interlock relay fail to close
	IF Devices.Coil[i].CloseACInterlockRly = TRUE AND Devices.Coil[i].AC_Interlock_RlyClose = FALSE AND Devices.Coil[i].CoilEnabled = TRUE THEN
		Trips_DB.Coil[i].ACintLockRlyCloseFaultDelay_TON (IN := TRUE, PT := ACintLockRlyFaultDelay_PT);
		ELSE
			Trips_DB.Coil[i].ACintLockRlyCloseFaultDelay_TON (IN := FALSE, PT := ACintLockRlyFaultDelay_PT);
	END_IF;
	IF Trips_DB.Coil[i].ACintLockRlyCloseFaultDelay_TON.Q = TRUE THEN
		Trips_DB.Coil[i].ACInterlockRelayFailedtoClose := TRUE;	
		Trips_DB.Coil[i].ACintLockRlyCloseFaultDelay_TON (IN := FALSE, PT := ACintLockRlyFaultDelay_PT);
	END_IF;
	
	//hv iso 
	IF Devices.Coil[i].CloseHVisolationRelay = TRUE AND Devices.Coil[i].HVisolationRelayClosed = FALSE AND Devices.Coil[i].CoilEnabled = TRUE THEN
		Trips_DB.Coil[i].HVRelayCloseFaultDelay_TON (IN := TRUE, PT := HVisoRlyFaultDelay_PT);
		ELSE
			Trips_DB.Coil[i].HVRelayCloseFaultDelay_TON (IN := FALSE, PT := HVisoRlyFaultDelay_PT);
	END_IF
	
	IF Trips_DB.Coil[i].HVRelayCloseFaultDelay_TON.Q = TRUE THEN
		Trips_DB.Coil[i].HVisoRelayFailedToClose := TRUE; 
		Trips_DB.Coil[i].HVRelayCloseFaultDelay_TON (IN := FALSE);
	END_IF;

	IF Devices.Coil[i].CloseHVisolationRelay = FALSE AND Devices.Coil[i].HVisolationRelayClosed = TRUE AND Devices.Coil[i].CoilEnabled = TRUE THEN
		Trips_DB.Coil[i].HVRelayOpenFaultDelay_TON (IN := TRUE, PT := HVisoRlyFaultDelay_PT);
		ELSE
			Trips_DB.Coil[i].HVRelayOpenFaultDelay_TON (IN := FALSE, PT := HVisoRlyFaultDelay_PT);
	END_IF
	
	IF Trips_DB.Coil[i].HVRelayOpenFaultDelay_TON.Q = TRUE THEN
		Trips_DB.Coil[i].HVisoRelayFailedToOpen := TRUE; 
		Trips_DB.Coil[i].HVRelayOpenFaultDelay_TON (IN := FALSE, PT := HVisoRlyFaultDelay_PT);
	END_IF
	
	//check to see if Dump relay failed to open
	IF Devices.Coil[i].OpenDumpRelays = TRUE AND 
		(Devices.Coil[i].DumpRelay1_closed = TRUE OR Devices.Coil[i].DumpRelay2_closed = TRUE) AND
		Devices.Coil[i].CoilEnabled = TRUE 
		THEN
			Trips_DB.Coil[i].DumpRlyOpenFaultDelay_TON (IN := TRUE, PT := DumpRly1FaultDelay_PT);
		ELSE
			Trips_DB.Coil[i].DumpRlyOpenFaultDelay_TON (IN := FALSE, PT := DumpRly1FaultDelay_PT);
	END_IF;
	IF Trips_DB.Coil[i].DumpRlyOpenFaultDelay_TON.Q = TRUE THEN
		Trips_DB.Coil[i].DumpRelay1_FailtoOpen := TRUE;
		Trips_DB.Coil[i].DumpRelay2_FailtoOpen := TRUE;
		Trips_DB.Coil[i].DumpRlyOpenFaultDelay_TON (IN := FALSE, PT := DumpRly1FaultDelay_PT);		
	END_IF;

	//check to see if charge relay failed to close
	IF Devices.Coil[i].closeChargeRelay = TRUE AND Devices.Coil[i].ChargeRelay_closed = FALSE AND Devices.Coil[i].CoilEnabled = TRUE THEN
		Trips_DB.Coil[i].ChrgRlyCloseFaultDelay_TON (IN := TRUE, PT := ChrgRlyFaultDelay_PT);
		ELSE
			Trips_DB.Coil[i].ChrgRlyCloseFaultDelay_TON (IN := FALSE, PT := ChrgRlyFaultDelay_PT);
		END_IF;
	IF Trips_DB.Coil[i].ChrgRlyCloseFaultDelay_TON.Q = TRUE THEN
		Trips_DB.Coil[i].ChargeRelay_FailtoClose := TRUE;
		Trips_DB.Coil[i].ChrgRlyCloseFaultDelay_TON (IN := FALSE, PT := ChrgRlyFaultDelay_PT);
	END_IF;

	//check to see if AC interlock relay fail to open
	IF Devices.Coil[i].CloseACInterlockRly = FALSE AND Devices.Coil[i].AC_Interlock_RlyClose = TRUE AND Devices.Coil[i].CoilEnabled = TRUE THEN
		Trips_DB.Coil[i].ACintLockRlyOpenFaultDelay_TON (IN := TRUE, PT := ACintLockRlyFaultDelay_PT);
		ELSE
			Trips_DB.Coil[i].ACintLockRlyOpenFaultDelay_TON (IN := FALSE, PT := ACintLockRlyFaultDelay_PT);
		END_IF;
	IF Trips_DB.Coil[i].ACintLockRlyOpenFaultDelay_TON.Q = TRUE THEN
		Trips_DB.Coil[i].ACInterlockRelayFailedtoOpen := TRUE;	
		Trips_DB.Coil[i].ACintLockRlyOpenFaultDelay_TON (IN := FALSE, PT := ACintLockRlyFaultDelay_PT);//debounce
	END_IF;
	
	//check to see if Dump relay failed to close
	IF Devices.Coil[i].OpenDumpRelays = FALSE AND 
		(Devices.Coil[i].DumpRelay1_closed = FALSE OR Devices.Coil[i].DumpRelay2_closed = FALSE) AND 
		Devices.Coil[i].CoilEnabled = TRUE 
		THEN
			Trips_DB.Coil[i].DumpRlyCloseFaultDelay_TON (IN := TRUE, PT := DumpRly1FaultDelay_PT);
		ELSE
			Trips_DB.Coil[i].DumpRlyCloseFaultDelay_TON (IN := FALSE, PT := DumpRly1FaultDelay_PT);
	END_IF;
	IF Trips_DB.Coil[i].DumpRlyCloseFaultDelay_TON.Q = TRUE THEN
		Trips_DB.Coil[i].DumpRelay1_FailtoClose := TRUE;
		Trips_DB.Coil[i].DumpRelay2_FailtoClose := TRUE;	
		Trips_DB.Coil[i].DumpRlyCloseFaultDelay_TON (IN := FALSE, PT := DumpRly1FaultDelay_PT);	
	END_IF;
	
	//check to see if charge relay failed to open
	IF Devices.Coil[i].closeChargeRelay = FALSE AND Devices.Coil[i].ChargeRelay_closed = TRUE AND Devices.Coil[i].CoilEnabled = TRUE THEN
		Trips_DB.Coil[i].ChrgRlyOpenFaultDelay_TON (IN := TRUE, PT := ChrgRlyFaultDelay_PT);
		ELSE
			Trips_DB.Coil[i].ChrgRlyOpenFaultDelay_TON (IN := FALSE, PT := ChrgRlyFaultDelay_PT);
		END_IF;
	IF Trips_DB.Coil[i].ChrgRlyOpenFaultDelay_TON.Q = TRUE THEN
		Trips_DB.Coil[i].ChargeRelay_FailtoOpen := TRUE;
		Trips_DB.Coil[i].ChrgRlyOpenFaultDelay_TON (IN := FALSE, PT := ChrgRlyFaultDelay_PT);
	END_IF;
	
	//Any Charge Relay fail to open or close
	IF Trips_DB.Coil[i].ChargeRelay_FailtoClose = TRUE OR Trips_DB.Coil[i].ChargeRelay_FailtoOpen = TRUE THEN
		Trips_DB.AnyChargeRlyFail := TRUE;
	END_IF;
	//Any Dump relay fail to open or close
	IF Trips_DB.Coil[i].DumpRelay1_FailtoClose = TRUE OR Trips_DB.Coil[i].DumpRelay1_FailtoOpen = TRUE OR 
		Trips_DB.Coil[i].DumpRelay2_FailtoClose = TRUE OR Trips_DB.Coil[i].DumpRelay2_FailtoOpen = TRUE
		THEN
			Trips_DB.AnyDumpRlyFail := TRUE;
	END_IF;
	//Any ac relay fail to open or close
	IF Trips_DB.Coil[i].ACInterlockRelayFailedtoClose = TRUE OR Trips_DB.Coil[i].ACInterlockRelayFailedtoOpen = TRUE
		THEN
			Trips_DB.AnyACInterlockFail := TRUE;
	END_IF;
	
	IF Trips_DB.Coil[i].HVisoRelayFailedToClose = TRUE OR Trips_DB.Coil[i].HVisoRelayFailedToOpen = TRUE THEN
		Trips_DB.AnyHVisoRelayFailed := TRUE;
	END_IF
END_FOR;	

//UC warnings and alarms
FOR i := 1 TO 10 BY 1 DO
	FOR j:= 1 TO 10 BY 1 DO 
		//over voltage
		IF Devices.Coil[i].UltraCap[j].Elec_OverVoltage = 1 THEN 
			Trips_DB.Coil[i].UltraCap[j].UC_Cell_OverV_warning := TRUE;
		ELSIF Devices.Coil[i].UltraCap[j].Elec_OverVoltage = 2 THEN
			Trips_DB.Coil[i].UltraCap[j].UC_Cell_OverV_alarm := TRUE;
		ELSIF Devices.Coil[i].UltraCap[1].Elec_OverVoltage = 0 THEN
			Trips_DB.Coil[i].UltraCap[j].UC_Cell_OverV_warning := FALSE;
			Trips_DB.Coil[i].UltraCap[j].UC_Cell_OverV_alarm := FALSE;
		END_IF
		
		//high temp
		IF Devices.Coil[i].UltraCap[j].Therm_HighTemp = 1 THEN 
			Trips_DB.Coil[i].UltraCap[j].UC_tempHigh_warning := TRUE;
		ELSIF Devices.Coil[i].UltraCap[j].Therm_HighTemp = 2 THEN
			Trips_DB.Coil[i].UltraCap[j].UC_tempHigh_alarm := TRUE;
		ELSIF Devices.Coil[i].UltraCap[j].Therm_HighTemp = 0 THEN 
			Trips_DB.Coil[i].UltraCap[j].UC_tempHigh_warning := FALSE;
			Trips_DB.Coil[i].UltraCap[j].UC_tempHigh_alarm := FALSE;
		END_IF;	
		
		//any cap overtemp warning
		IF Trips_DB.Coil[i].UltraCap[j].UC_tempHigh_warning = TRUE THEN
			Trips_DB.Coil[i].AnyCapOverTemp_warning := TRUE;
			ELSE
				Trips_DB.Coil[i].AnyCapOverTemp_warning := FALSE;
		END_IF;
		//any cap overtemp alarm
		IF Trips_DB.Coil[i].UltraCap[j].UC_tempHigh_alarm = TRUE THEN
			Trips_DB.Coil[i].AnyCapOverTemp_alarm := TRUE;
			ELSE
				Trips_DB.Coil[i].AnyCapOverTemp_alarm := FALSE;
		END_IF;
		
		//any cap over voltage warning
		IF Trips_DB.Coil[i].UltraCap[j].UC_Cell_OverV_warning = TRUE THEN
			Trips_DB.Coil[i].AnyCapOverV_warning := TRUE;
			ELSE 
				Trips_DB.Coil[i].AnyCapOverV_warning := FALSE;
		END_IF
		
		//any cap over voltage alarm
		IF Trips_DB.Coil[i].UltraCap[j].UC_Cell_OverV_alarm = TRUE THEN
			Trips_DB.Coil[i].AnyCapOverV_alarm := TRUE;
			ELSE 
				Trips_DB.Coil[i].AnyCapOverV_alarm := FALSE;
		END_IF
		
		//any coil cap warning
		IF Trips_DB.Coil[i].AnyCapOverV_warning = TRUE OR Trips_DB.Coil[i].AnyCapOverTemp_warning = TRUE THEN
			Devices.Coil[i].CapWarning := TRUE;  //used for charge pause permissives
			ELSE
				Devices.Coil[i].CapWarning := FALSE;
		END_IF;
		
		//any coil cap alarm
		IF Trips_DB.Coil[i].AnyCapOverV_alarm = TRUE OR Trips_DB.Coil[i].AnyCapOverTemp_alarm = TRUE THEN
			Devices.Coil[i].CapAlarm := TRUE;  //ussed for charge pause permissives
			ELSE
				Devices.Coil[i].CapAlarm := FALSE;
		END_IF
		
	END_FOR
END_FOR


//*******************E-Stop Trips
FOR i := 1 TO 10 DO 
	IF Devices.Coil[i].Local_StopPB_Pressed = TRUE OR MCP_IO.MasterStopPB_Pressed = TRUE THEN
		Trips_DB.AnyEstopPressed := TRUE;
	END_IF;	
END_FOR;

FOR i := 1 TO 10 BY 1 DO
	IF (Trips_DB.Coil[i].ACInterlockRelayFailedtoClose = TRUE OR 
		Trips_DB.Coil[i].ACInterlockRelayFailedtoOpen = TRUE OR 
		Trips_DB.Coil[i].HVisoRelayFailedToClose = TRUE OR 
		Trips_DB.Coil[i].HVisoRelayFailedToOpen = TRUE OR
		Trips_DB.Coil[i].ChargeRelay_FailtoClose = TRUE OR
		Trips_DB.Coil[i].ChargeRelay_FailtoOpen = TRUE OR
		Trips_DB.Coil[i].DumpRelay1_FailtoClose =  TRUE OR 
		Trips_DB.Coil[i].DumpRelay1_FailtoOpen = TRUE OR 
		Trips_DB.Coil[i].DumpRelay2_FailtoClose =  TRUE OR 
		Trips_DB.Coil[i].DumpRelay2_FailtoOpen = TRUE OR 
		Trips_DB.Coil[i].ChargerVoltageReadingFaulted = TRUE OR
		Trips_DB.Coil[i].CurrentReadingFaulted = TRUE OR
		Devices.Coil[i].Local_StopPB_Pressed = TRUE OR
		Devices.Coil[i].LossPneumaticPressure = FALSE) AND Devices.Coil[i].CoilEnabled = TRUE 	
		THEN
			Devices.Coil[i].SystemFaulted := TRUE;
	END_IF
	
	IF Devices.Coil[i].SystemFaulted = TRUE THEN
		Trips_DB.SystemTripped := TRUE;
	END_IF;
END_FOR;

//timer runout


//*********************************** Test
(*IF InstrumentReading.R2_01_CH01 <= 0.0 THEN
	delay2s(input := FALSE);
ELSE 
	delay2s (input := TRUE);
END_IF;
bTest := delay2s.output;
*)
// Instrumentation Hardware trip
//Input.R2_01_00_Status.0;

//************** Clear System Fault
IF GVL.ClearAllFaults = TRUE OR stControl.ClearAllFault = TRUE THEN
	Trips_DB.InstrumentationFaulted := FALSE;
	Trips_DB.SystemTripped := FALSE;
	Trips_DB.AnyEstopPressed := FALSE;
	Trips_DB.AnyDumpRlyFail := FALSE;
	Trips_DB.AnyChargeRlyFail := FALSE;
	Trips_DB.AnyACInterlockFail := FALSE;
	
	Trips_DB.AnyDCPSU_fail := FALSE;
	Trips_DB.AnyHVisoRelayFailed := FALSE;
	Trips_DB.MachineTimedOut := FALSE;
	
	//reset relay trips
	FOR i := 1 TO 10 BY 1 DO 
		Trips_DB.Coil[i].ACInterlockRelayFailedtoClose := FALSE;
		Trips_DB.Coil[i].ACInterlockRelayFailedtoOpen := FALSE;
		Trips_DB.Coil[i].DumpRelay1_FailtoClose := FALSE;
		Trips_DB.Coil[i].DumpRelay1_FailtoOpen := FALSE;
		Trips_DB.Coil[i].DumpRelay2_FailtoClose := FALSE;
		Trips_DB.Coil[i].DumpRelay2_FailtoOpen := FALSE;
		Trips_DB.Coil[i].ChargeRelay_FailtoClose := FALSE;
		Trips_DB.Coil[i].ChargeRelay_FailtoOpen := FALSE;
		Devices.Coil[i].SystemFaulted := FALSE; 
		
		Trips_DB.Coil[i].HVisoRelayFailedToOpen := FALSE;
		Trips_DB.Coil[i].HVisoRelayFailedToClose := FALSE;
		
		FOR j := 1 TO 10 BY 1 DO
			Trips_DB.Coil[i].UltraCap[j].UC_Cell_OverV_alarm := FALSE;
			Trips_DB.Coil[i].UltraCap[j].UC_tempHigh_alarm := FALSE;
			Trips_DB.Coil[i].UltraCap[j].UC_Cell_OverV_warning := FALSE;
			Trips_DB.Coil[i].UltraCap[j].UC_tempHigh_warning := FALSE;
		END_FOR;
	END_FOR;
	
	evtLogger.ClearAllAlarms(0, FALSE);
	//evtLogger.ClearLoggedEvents(1);
END_IF;


IF i > 10 THEN 
	i := 1;
END_IF;

IF j > 10 THEN //will be 15 at full scale
	j := 1;
END_IF;

END_PROGRAM
